//     PlcTask Inputs/GVL_iXlinker.EtherCAT_Master_EJxxxx.Beckhoff_EJ3xxx.A_0016_EJ3202_0000_0021.RTD_Inputs_Channel_2.Status/Limit_2 <-> RTD Inputs Channel 2/Status/Limit 2
//     PlcTask Inputs/GVL_iXlinker.EtherCAT_Master_EJxxxx.Beckhoff_EJ3xxx.A_0016_EJ3202_0000_0021.RTD_Inputs_Channel_1.Status/Error <-> RTD Inputs Channel 1/Status/Error
//     PlcTask Inputs/GVL_iXlinker.EtherCAT_Master_EJxxxx.Beckhoff_EJ3xxx.A_0016_EJ3202_0000_0021.RTD_Inputs_Channel_2.Status/Error <-> RTD Inputs Channel 2/Status/Error
//     PlcTask Inputs/GVL_iXlinker.EtherCAT_Master_EJxxxx.Beckhoff_EJ3xxx.A_0016_EJ3202_0000_0021.RTD_Inputs_Channel_1.Status/TxPDO_State <-> RTD Inputs Channel 1/Status/TxPDO State
//     PlcTask Inputs/GVL_iXlinker.EtherCAT_Master_EJxxxx.Beckhoff_EJ3xxx.A_0016_EJ3202_0000_0021.RTD_Inputs_Channel_2.Status/TxPDO_State <-> RTD Inputs Channel 2/Status/TxPDO State
//     PlcTask Inputs/GVL_iXlinker.EtherCAT_Master_EJxxxx.Beckhoff_EJ3xxx.A_0016_EJ3202_0000_0021.RTD_Inputs_Channel_1.Status/TxPDO_Toggle <-> RTD Inputs Channel 1/Status/TxPDO Toggle
//     PlcTask Inputs/GVL_iXlinker.EtherCAT_Master_EJxxxx.Beckhoff_EJ3xxx.A_0016_EJ3202_0000_0021.RTD_Inputs_Channel_2.Status/TxPDO_Toggle <-> RTD Inputs Channel 2/Status/TxPDO Toggle
//     PlcTask Inputs/GVL_iXlinker.EtherCAT_Master_EJxxxx.Beckhoff_EJ3xxx.A_0016_EJ3202_0000_0021.RTD_Inputs_Channel_1.Value <-> RTD Inputs Channel 1/Value
//     PlcTask Inputs/GVL_iXlinker.EtherCAT_Master_EJxxxx.Beckhoff_EJ3xxx.A_0016_EJ3202_0000_0021.RTD_Inputs_Channel_2.Value <-> RTD Inputs Channel 2/Value
//     PlcTask Inputs/GVL_iXlinker.EtherCAT_Master_EJxxxx.Beckhoff_EJ3xxx.A_0016_EJ3202_0000_0021.WcState.WcState <-> WcState/WcState
//     PlcTask Inputs/GVL_iXlinker.EtherCAT_Master_EJxxxx.Beckhoff_EJ3xxx.A_0016_EJ3202_0000_0021.WcState.InputToggle <-> WcState/InputToggle
//     PlcTask Inputs/GVL_iXlinker.EtherCAT_Master_EJxxxx.Beckhoff_EJ3xxx.A_0016_EJ3202_0000_0021.InfoData.AdsAddr <-> InfoData/AdsAddr
//     PlcTask Inputs/GVL_iXlinker.EtherCAT_Master_EJxxxx.Beckhoff_EJ3xxx.A_0016_EJ3202_0000_0021.InfoData.State <-> InfoData/State
//   PLC/PLC Instance <-> EtherCAT Master EJxxxx/Beckhoff EJ3xxx/A_0017(EJ3214-0000-0016)
//     PlcTask Inputs/GVL_iXlinker.EtherCAT_Master_EJxxxx.Beckhoff_EJ3xxx.A_0017_EJ3214_0000_0016.RTD_Inputs_Channel_1.Status/Underrange <-> RTD Inputs Channel 1/Status/Underrange
//     PlcTask Inputs/GVL_iXlinker.EtherCAT_Master_EJxxxx.Beckhoff_EJ3xxx.A_0017_EJ3214_0000_0016.RTD_Inputs_Channel_2.Status/Underrange <-> RTD Inputs Channel 2/Status/Underrange
//     PlcTask Inputs/GVL_iXlinker.EtherCAT_Master_EJxxxx.Beckhoff_EJ3xxx.A_0017_EJ3214_0000_0016.RTD_Inputs_Channel_3.Status/Underrange <-> RTD Inputs Channel 3/Status/Underrange
//     PlcTask Inputs/GVL_iXlinker.EtherCAT_Master_EJxxxx.Beckhoff_EJ3xxx.A_0017_EJ3214_0000_0016.RTD_Inputs_Channel_4.Status/Underrange <-> RTD Inputs Channel 4/Status/Underrange
//     PlcTask Inputs/GVL_iXlinker.EtherCAT_Master_EJxxxx.Beckhoff_EJ3xxx.A_0017_EJ3214_0000_0016.RTD_Inputs_Channel_1.Status/Overrange <-> RTD Inputs Channel 1/Status/Overrange
//     PlcTask Inputs/GVL_iXlinker.EtherCAT_Master_EJxxxx.Beckhoff_EJ3xxx.A_0017_EJ3214_0000_0016.RTD_Inputs_Channel_2.Status/Overrange <-> RTD Inputs Channel 2/Status/Overrange
//     PlcTask Inputs/GVL_iXlinker.EtherCAT_Master_EJxxxx.Beckhoff_EJ3xxx.A_0017_EJ3214_0000_0016.RTD_Inputs_Channel_3.Status/Overrange <-> RTD Inputs Channel 3/Status/Overrange
//     PlcTask Inputs/GVL_iXlinker.EtherCAT_Master_EJxxxx.Beckhoff_EJ3xxx.A_0017_EJ3214_0000_0016.RTD_Inputs_Channel_4.Status/Overrange <-> RTD Inputs Channel 4/Status/Overrange
//     PlcTask Inputs/GVL_iXlinker.EtherCAT_Master_EJxxxx.Beckhoff_EJ3xxx.A_0017_EJ3214_0000_0016.RTD_Inputs_Channel_1.Status/Error <-> RTD Inputs Channel 1/Status/Error
//     PlcTask Inputs/GVL_iXlinker.EtherCAT_Master_EJxxxx.Beckhoff_EJ3xxx.A_0017_EJ3214_0000_0016.RTD_Inputs_Channel_2.Status/Error <-> RTD Inputs Channel 2/Status/Error
//     PlcTask Inputs/GVL_iXlinker.EtherCAT_Master_EJxxxx.Beckhoff_EJ3xxx.A_0017_EJ3214_0000_0016.RTD_Inputs_Channel_3.Status/Error <-> RTD Inputs Channel 3/Status/Error
//     PlcTask Inputs/GVL_iXlinker.EtherCAT_Master_EJxxxx.Beckhoff_EJ3xxx.A_0017_EJ3214_0000_0016.RTD_Inputs_Channel_4.Status/Error <-> RTD Inputs Channel 4/Status/Error
//     PlcTask Inputs/GVL_iXlinker.EtherCAT_Master_EJxxxx.Beckhoff_EJ3xxx.A_0017_EJ3214_0000_0016.RTD_Inputs_Channel_1.Status/TxPDO_State <-> RTD Inputs Channel 1/Status/TxPDO State
//     PlcTask Inputs/GVL_iXlinker.EtherCAT_Master_EJxxxx.Beckhoff_EJ3xxx.A_0017_EJ3214_0000_0016.RTD_Inputs_Channel_2.Status/TxPDO_State <-> RTD Inputs Channel 2/Status/TxPDO State
//     PlcTask Inputs/GVL_iXlinker.EtherCAT_Master_EJxxxx.Beckhoff_EJ3xxx.A_0017_EJ3214_0000_0016.RTD_Inputs_Channel_3.Status/TxPDO_State <-> RTD Inputs Channel 3/Status/TxPDO State
//     PlcTask Inputs/GVL_iXlinker.EtherCAT_Master_EJxxxx.Beckhoff_EJ3xxx.A_0017_EJ3214_0000_0016.RTD_Inputs_Channel_4.Status/TxPDO_State <-> RTD Inputs Channel 4/Status/TxPDO State
//     PlcTask Inputs/GVL_iXlinker.EtherCAT_Master_EJxxxx.Beckhoff_EJ3xxx.A_0017_EJ3214_0000_0016.RTD_Inputs_Channel_1.Status/TxPDO_Toggle <-> RTD Inputs Channel 1/Status/TxPDO Toggle
//     PlcTask Inputs/GVL_iXlinker.EtherCAT_Master_EJxxxx.Beckhoff_EJ3xxx.A_0017_EJ3214_0000_0016.RTD_Inputs_Channel_2.Status/TxPDO_Toggle <-> RTD Inputs Channel 2/Status/TxPDO Toggle
//     PlcTask Inputs/GVL_iXlinker.EtherCAT_Master_EJxxxx.Beckhoff_EJ3xxx.A_0017_EJ3214_0000_0016.RTD_Inputs_Channel_3.Status/TxPDO_Toggle <-> RTD Inputs Channel 3/Status/TxPDO Toggle
//     PlcTask Inputs/GVL_iXlinker.EtherCAT_Master_EJxxxx.Beckhoff_EJ3xxx.A_0017_EJ3214_0000_0016.RTD_Inputs_Channel_4.Status/TxPDO_Toggle <-> RTD Inputs Channel 4/Status/TxPDO Toggle
//     PlcTask Inputs/GVL_iXlinker.EtherCAT_Master_EJxxxx.Beckhoff_EJ3xxx.A_0017_EJ3214_0000_0016.RTD_Inputs_Channel_1.Value <-> RTD Inputs Channel 1/Value
//     PlcTask Inputs/GVL_iXlinker.EtherCAT_Master_EJxxxx.Beckhoff_EJ3xxx.A_0017_EJ3214_0000_0016.RTD_Inputs_Channel_2.Value <-> RTD Inputs Channel 2/Value
//     PlcTask Inputs/GVL_iXlinker.EtherCAT_Master_EJxxxx.Beckhoff_EJ3xxx.A_0017_EJ3214_0000_0016.RTD_Inputs_Channel_3.Value <-> RTD Inputs Channel 3/Value
//     PlcTask Inputs/GVL_iXlinker.EtherCAT_Master_EJxxxx.Beckhoff_EJ3xxx.A_0017_EJ3214_0000_0016.RTD_Inputs_Channel_4.Value <-> RTD Inputs Channel 4/Value
//     PlcTask Inputs/GVL_iXlinker.EtherCAT_Master_EJxxxx.Beckhoff_EJ3xxx.A_0017_EJ3214_0000_0016.WcState.WcState <-> WcState/WcState
//     PlcTask Inputs/GVL_iXlinker.EtherCAT_Master_EJxxxx.Beckhoff_EJ3xxx.A_0017_EJ3214_0000_0016.WcState.InputToggle <-> WcState/InputToggle
//     PlcTask Inputs/GVL_iXlinker.EtherCAT_Master_EJxxxx.Beckhoff_EJ3xxx.A_0017_EJ3214_0000_0016.InfoData.AdsAddr <-> InfoData/AdsAddr
//     PlcTask Inputs/GVL_iXlinker.EtherCAT_Master_EJxxxx.Beckhoff_EJ3xxx.A_0017_EJ3214_0000_0016.InfoData.State <-> InfoData/State
//   PLC/PLC Instance <-> EtherCAT Master EJxxxx/Beckhoff EJ3xxx/A_0018(EJ3255-0000-0023)
//     PlcTask Inputs/GVL_iXlinker.EtherCAT_Master_EJxxxx.Beckhoff_EJ3xxx.A_0018_EJ3255_0000_0023.AI_Standard_Channel_1.Status/Underrange <-> AI Standard Channel 1/Status/Underrange
//     PlcTask Inputs/GVL_iXlinker.EtherCAT_Master_EJxxxx.Beckhoff_EJ3xxx.A_0018_EJ3255_0000_0023.AI_Standard_Channel_2.Status/Underrange <-> AI Standard Channel 2/Status/Underrange
//     PlcTask Inputs/GVL_iXlinker.EtherCAT_Master_EJxxxx.Beckhoff_EJ3xxx.A_0018_EJ3255_0000_0023.AI_Standard_Channel_3.Status/Underrange <-> AI Standard Channel 3/Status/Underrange
//     PlcTask Inputs/GVL_iXlinker.EtherCAT_Master_EJxxxx.Beckhoff_EJ3xxx.A_0018_EJ3255_0000_0023.AI_Standard_Channel_4.Status/Underrange <-> AI Standard Channel 4/Status/Underrange
//     PlcTask Inputs/GVL_iXlinker.EtherCAT_Master_EJxxxx.Beckhoff_EJ3xxx.A_0018_EJ3255_0000_0023.AI_Standard_Channel_5.Status/Underrange <-> AI Standard Channel 5/Status/Underrange
//     PlcTask Inputs/GVL_iXlinker.EtherCAT_Master_EJxxxx.Beckhoff_EJ3xxx.A_0018_EJ3255_0000_0023.AI_Standard_Channel_1.Status/Overrange <-> AI Standard Channel 1/Status/Overrange
//     PlcTask Inputs/GVL_iXlinker.EtherCAT_Master_EJxxxx.Beckhoff_EJ3xxx.A_0018_EJ3255_0000_0023.AI_Standard_Channel_2.Status/Overrange <-> AI Standard Channel 2/Status/Overrange
//     PlcTask Inputs/GVL_iXlinker.EtherCAT_Master_EJxxxx.Beckhoff_EJ3xxx.A_0018_EJ3255_0000_0023.AI_Standard_Channel_3.Status/Overrange <-> AI Standard Channel 3/Status/Overrange
//     PlcTask Inputs/GVL_iXlinker.EtherCAT_Master_EJxxxx.Beckhoff_EJ3xxx.A_0018_EJ3255_0000_0023.AI_Standard_Channel_4.Status/Overrange <-> AI Standard Channel 4/Status/Overrange
//     PlcTask Inputs/GVL_iXlinker.EtherCAT_Master_EJxxxx.Beckhoff_EJ3xxx.A_0018_EJ3255_0000_0023.AI_Standard_Channel_5.Status/Overrange <-> AI Standard Channel 5/Status/Overrange
//     PlcTask Inputs/GVL_iXlinker.EtherCAT_Master_EJxxxx.Beckhoff_EJ3xxx.A_0018_EJ3255_0000_0023.AI_Standard_Channel_1.Status/Limit_1 <-> AI Standard Channel 1/Status/Limit 1
//     PlcTask Inputs/GVL_iXlinker.EtherCAT_Master_EJxxxx.Beckhoff_EJ3xxx.A_0018_EJ3255_0000_0023.AI_Standard_Channel_1.Status/Limit_2 <-> AI Standard Channel 1/Status/Limit 2
//     PlcTask Inputs/GVL_iXlinker.EtherCAT_Master_EJxxxx.Beckhoff_EJ3xxx.A_0018_EJ3255_0000_0023.AI_Standard_Channel_2.Status/Limit_1 <-> AI Standard Channel 2/Status/Limit 1
//     PlcTask Inputs/GVL_iXlinker.EtherCAT_Master_EJxxxx.Beckhoff_EJ3xxx.A_0018_EJ3255_0000_0023.AI_Standard_Channel_2.Status/Limit_2 <-> AI Standard Channel 2/Status/Limit 2
//     PlcTask Inputs/GVL_iXlinker.EtherCAT_Master_EJxxxx.Beckhoff_EJ3xxx.A_0018_EJ3255_0000_0023.AI_Standard_Channel_3.Status/Limit_1 <-> AI Standard Channel 3/Status/Limit 1
//     PlcTask Inputs/GVL_iXlinker.EtherCAT_Master_EJxxxx.Beckhoff_EJ3xxx.A_0018_EJ3255_0000_0023.AI_Standard_Channel_3.Status/Limit_2 <-> AI Standard Channel 3/Status/Limit 2
//     PlcTask Inputs/GVL_iXlinker.EtherCAT_Master_EJxxxx.Beckhoff_EJ3xxx.A_0018_EJ3255_0000_0023.AI_Standard_Channel_4.Status/Limit_1 <-> AI Standard Channel 4/Status/Limit 1
//     PlcTask Inputs/GVL_iXlinker.EtherCAT_Master_EJxxxx.Beckhoff_EJ3xxx.A_0018_EJ3255_0000_0023.AI_Standard_Channel_4.Status/Limit_2 <-> AI Standard Channel 4/Status/Limit 2
//     PlcTask Inputs/GVL_iXlinker.EtherCAT_Master_EJxxxx.Beckhoff_EJ3xxx.A_0018_EJ3255_0000_0023.AI_Standard_Channel_5.Status/Limit_1 <-> AI Standard Channel 5/Status/Limit 1
//     PlcTask Inputs/GVL_iXlinker.EtherCAT_Master_EJxxxx.Beckhoff_EJ3xxx.A_0018_EJ3255_0000_0023.AI_Standard_Channel_5.Status/Limit_2 <-> AI Standard Channel 5/Status/Limit 2
//     PlcTask Inputs/GVL_iXlinker.EtherCAT_Master_EJxxxx.Beckhoff_EJ3xxx.A_0018_EJ3255_0000_0023.AI_Standard_Channel_1.Status/Error <-> AI Standard Channel 1/Status/Error
//     PlcTask Inputs/GVL_iXlinker.EtherCAT_Master_EJxxxx.Beckhoff_EJ3xxx.A_0018_EJ3255_0000_0023.AI_Standard_Channel_2.Status/Error <-> AI Standard Channel 2/Status/Error
//     PlcTask Inputs/GVL_iXlinker.EtherCAT_Master_EJxxxx.Beckhoff_EJ3xxx.A_0018_EJ3255_0000_0023.AI_Standard_Channel_3.Status/Error <-> AI Standard Channel 3/Status/Error
//     PlcTask Inputs/GVL_iXlinker.EtherCAT_Master_EJxxxx.Beckhoff_EJ3xxx.A_0018_EJ3255_0000_0023.AI_Standard_Channel_4.Status/Error <-> AI Standard Channel 4/Status/Error
//     PlcTask Inputs/GVL_iXlinker.EtherCAT_Master_EJxxxx.Beckhoff_EJ3xxx.A_0018_EJ3255_0000_0023.AI_Standard_Channel_5.Status/Error <-> AI Standard Channel 5/Status/Error
//     PlcTask Inputs/GVL_iXlinker.EtherCAT_Master_EJxxxx.Beckhoff_EJ3xxx.A_0018_EJ3255_0000_0023.AI_Standard_Channel_1.Status/Sync_error <-> AI Standard Channel 1/Status/Sync error
//     PlcTask Inputs/GVL_iXlinker.EtherCAT_Master_EJxxxx.Beckhoff_EJ3xxx.A_0018_EJ3255_0000_0023.AI_Standard_Channel_2.Status/Sync_error <-> AI Standard Channel 2/Status/Sync error
//     PlcTask Inputs/GVL_iXlinker.EtherCAT_Master_EJxxxx.Beckhoff_EJ3xxx.A_0018_EJ3255_0000_0023.AI_Standard_Channel_3.Status/Sync_error <-> AI Standard Channel 3/Status/Sync error
//     PlcTask Inputs/GVL_iXlinker.EtherCAT_Master_EJxxxx.Beckhoff_EJ3xxx.A_0018_EJ3255_0000_0023.AI_Standard_Channel_4.Status/Sync_error <-> AI Standard Channel 4/Status/Sync error
//     PlcTask Inputs/GVL_iXlinker.EtherCAT_Master_EJxxxx.Beckhoff_EJ3xxx.A_0018_EJ3255_0000_0023.AI_Standard_Channel_5.Status/Sync_error <-> AI Standard Channel 5/Status/Sync error
//     PlcTask Inputs/GVL_iXlinker.EtherCAT_Master_EJxxxx.Beckhoff_EJ3xxx.A_0018_EJ3255_0000_0023.AI_Standard_Channel_1.Status/TxPDO_State <-> AI Standard Channel 1/Status/TxPDO State
//     PlcTask Inputs/GVL_iXlinker.EtherCAT_Master_EJxxxx.Beckhoff_EJ3xxx.A_0018_EJ3255_0000_0023.AI_Standard_Channel_2.Status/TxPDO_State <-> AI Standard Channel 2/Status/TxPDO State
//     PlcTask Inputs/GVL_iXlinker.EtherCAT_Master_EJxxxx.Beckhoff_EJ3xxx.A_0018_EJ3255_0000_0023.AI_Standard_Channel_3.Status/TxPDO_State <-> AI Standard Channel 3/Status/TxPDO State
//     PlcTask Inputs/GVL_iXlinker.EtherCAT_Master_EJxxxx.Beckhoff_EJ3xxx.A_0018_EJ3255_0000_0023.AI_Standard_Channel_4.Status/TxPDO_State <-> AI Standard Channel 4/Status/TxPDO State
//     PlcTask Inputs/GVL_iXlinker.EtherCAT_Master_EJxxxx.Beckhoff_EJ3xxx.A_0018_EJ3255_0000_0023.AI_Standard_Channel_5.Status/TxPDO_State <-> AI Standard Channel 5/Status/TxPDO State
//     PlcTask Inputs/GVL_iXlinker.EtherCAT_Master_EJxxxx.Beckhoff_EJ3xxx.A_0018_EJ3255_0000_0023.AI_Standard_Channel_1.Status/TxPDO_Toggle <-> AI Standard Channel 1/Status/TxPDO Toggle
//     PlcTask Inputs/GVL_iXlinker.EtherCAT_Master_EJxxxx.Beckhoff_EJ3xxx.A_0018_EJ3255_0000_0023.AI_Standard_Channel_2.Status/TxPDO_Toggle <-> AI Standard Channel 2/Status/TxPDO Toggle
//     PlcTask Inputs/GVL_iXlinker.EtherCAT_Master_EJxxxx.Beckhoff_EJ3xxx.A_0018_EJ3255_0000_0023.AI_Standard_Channel_3.Status/TxPDO_Toggle <-> AI Standard Channel 3/Status/TxPDO Toggle
//     PlcTask Inputs/GVL_iXlinker.EtherCAT_Master_EJxxxx.Beckhoff_EJ3xxx.A_0018_EJ3255_0000_0023.AI_Standard_Channel_4.Status/TxPDO_Toggle <-> AI Standard Channel 4/Status/TxPDO Toggle
//     PlcTask Inputs/GVL_iXlinker.EtherCAT_Master_EJxxxx.Beckhoff_EJ3xxx.A_0018_EJ3255_0000_0023.AI_Standard_Channel_5.Status/TxPDO_Toggle <-> AI Standard Channel 5/Status/TxPDO Toggle
//     PlcTask Inputs/GVL_iXlinker.EtherCAT_Master_EJxxxx.Beckhoff_EJ3xxx.A_0018_EJ3255_0000_0023.AI_Standard_Channel_1.Value <-> AI Standard Channel 1/Value
//     PlcTask Inputs/GVL_iXlinker.EtherCAT_Master_EJxxxx.Beckhoff_EJ3xxx.A_0018_EJ3255_0000_0023.AI_Standard_Channel_2.Value <-> AI Standard Channel 2/Value
//     PlcTask Inputs/GVL_iXlinker.EtherCAT_Master_EJxxxx.Beckhoff_EJ3xxx.A_0018_EJ3255_0000_0023.AI_Standard_Channel_3.Value <-> AI Standard Channel 3/Value
//     PlcTask Inputs/GVL_iXlinker.EtherCAT_Master_EJxxxx.Beckhoff_EJ3xxx.A_0018_EJ3255_0000_0023.AI_Standard_Channel_4.Value <-> AI Standard Channel 4/Value
//     PlcTask Inputs/GVL_iXlinker.EtherCAT_Master_EJxxxx.Beckhoff_EJ3xxx.A_0018_EJ3255_0000_0023.AI_Standard_Channel_5.Value <-> AI Standard Channel 5/Value
//     PlcTask Inputs/GVL_iXlinker.EtherCAT_Master_EJxxxx.Beckhoff_EJ3xxx.A_0018_EJ3255_0000_0023.WcState.WcState <-> WcState/WcState
//     PlcTask Inputs/GVL_iXlinker.EtherCAT_Master_EJxxxx.Beckhoff_EJ3xxx.A_0018_EJ3255_0000_0023.WcState.InputToggle <-> WcState/InputToggle
//     PlcTask Inputs/GVL_iXlinker.EtherCAT_Master_EJxxxx.Beckhoff_EJ3xxx.A_0018_EJ3255_0000_0023.InfoData.AdsAddr <-> InfoData/AdsAddr
//     PlcTask Inputs/GVL_iXlinker.EtherCAT_Master_EJxxxx.Beckhoff_EJ3xxx.A_0018_EJ3255_0000_0023.InfoData.State <-> InfoData/State
//   PLC/PLC Instance <-> EtherCAT Master EJxxxx/Beckhoff EJ3xxx/A_0019(EJ3318-0000-0017)
//     PlcTask Inputs/GVL_iXlinker.EtherCAT_Master_EJxxxx.Beckhoff_EJ3xxx.A_0019_EJ3318_0000_0017.TC_Channel_1.Status/Underrange <-> TC Channel 1/Status/Underrange
//     PlcTask Inputs/GVL_iXlinker.EtherCAT_Master_EJxxxx.Beckhoff_EJ3xxx.A_0019_EJ3318_0000_0017.TC_Channel_2.Status/Underrange <-> TC Channel 2/Status/Underrange
//     PlcTask Inputs/GVL_iXlinker.EtherCAT_Master_EJxxxx.Beckhoff_EJ3xxx.A_0019_EJ3318_0000_0017.TC_Channel_3.Status/Underrange <-> TC Channel 3/Status/Underrange
//     PlcTask Inputs/GVL_iXlinker.EtherCAT_Master_EJxxxx.Beckhoff_EJ3xxx.A_0019_EJ3318_0000_0017.TC_Channel_4.Status/Underrange <-> TC Channel 4/Status/Underrange
//     PlcTask Inputs/GVL_iXlinker.EtherCAT_Master_EJxxxx.Beckhoff_EJ3xxx.A_0019_EJ3318_0000_0017.TC_Channel_5.Status/Underrange <-> TC Channel 5/Status/Underrange
//     PlcTask Inputs/GVL_iXlinker.EtherCAT_Master_EJxxxx.Beckhoff_EJ3xxx.A_0019_EJ3318_0000_0017.TC_Channel_6.Status/Underrange <-> TC Channel 6/Status/Underrange
//     PlcTask Inputs/GVL_iXlinker.EtherCAT_Master_EJxxxx.Beckhoff_EJ3xxx.A_0019_EJ3318_0000_0017.TC_Channel_7.Status/Underrange <-> TC Channel 7/Status/Underrange
//     PlcTask Inputs/GVL_iXlinker.EtherCAT_Master_EJxxxx.Beckhoff_EJ3xxx.A_0019_EJ3318_0000_0017.TC_Channel_8.Status/Underrange <-> TC Channel 8/Status/Underrange
//     PlcTask Inputs/GVL_iXlinker.EtherCAT_Master_EJxxxx.Beckhoff_EJ3xxx.A_0019_EJ3318_0000_0017.TC_Channel_1.Status/Overrange <-> TC Channel 1/Status/Overrange
//     PlcTask Inputs/GVL_iXlinker.EtherCAT_Master_EJxxxx.Beckhoff_EJ3xxx.A_0019_EJ3318_0000_0017.TC_Channel_2.Status/Overrange <-> TC Channel 2/Status/Overrange
//     PlcTask Inputs/GVL_iXlinker.EtherCAT_Master_EJxxxx.Beckhoff_EJ3xxx.A_0019_EJ3318_0000_0017.TC_Channel_3.Status/Overrange <-> TC Channel 3/Status/Overrange
//     PlcTask Inputs/GVL_iXlinker.EtherCAT_Master_EJxxxx.Beckhoff_EJ3xxx.A_0019_EJ3318_0000_0017.TC_Channel_4.Status/Overrange <-> TC Channel 4/Status/Overrange
//     PlcTask Inputs/GVL_iXlinker.EtherCAT_Master_EJxxxx.Beckhoff_EJ3xxx.A_0019_EJ3318_0000_0017.TC_Channel_5.Status/Overrange <-> TC Channel 5/Status/Overrange
//     PlcTask Inputs/GVL_iXlinker.EtherCAT_Master_EJxxxx.Beckhoff_EJ3xxx.A_0019_EJ3318_0000_0017.TC_Channel_6.Status/Overrange <-> TC Channel 6/Status/Overrange
//     PlcTask Inputs/GVL_iXlinker.EtherCAT_Master_EJxxxx.Beckhoff_EJ3xxx.A_0019_EJ3318_0000_0017.TC_Channel_7.Status/Overrange <-> TC Channel 7/Status/Overrange
//     PlcTask Inputs/GVL_iXlinker.EtherCAT_Master_EJxxxx.Beckhoff_EJ3xxx.A_0019_EJ3318_0000_0017.TC_Channel_8.Status/Overrange <-> TC Channel 8/Status/Overrange
//     PlcTask Inputs/GVL_iXlinker.EtherCAT_Master_EJxxxx.Beckhoff_EJ3xxx.A_0019_EJ3318_0000_0017.TC_Channel_1.Status/Error <-> TC Channel 1/Status/Error
//     PlcTask Inputs/GVL_iXlinker.EtherCAT_Master_EJxxxx.Beckhoff_EJ3xxx.A_0019_EJ3318_0000_0017.TC_Channel_2.Status/Error <-> TC Channel 2/Status/Error
//     PlcTask Inputs/GVL_iXlinker.EtherCAT_Master_EJxxxx.Beckhoff_EJ3xxx.A_0019_EJ3318_0000_0017.TC_Channel_3.Status/Error <-> TC Channel 3/Status/Error
//     PlcTask Inputs/GVL_iXlinker.EtherCAT_Master_EJxxxx.Beckhoff_EJ3xxx.A_0019_EJ3318_0000_0017.TC_Channel_4.Status/Error <-> TC Channel 4/Status/Error
//     PlcTask Inputs/GVL_iXlinker.EtherCAT_Master_EJxxxx.Beckhoff_EJ3xxx.A_0019_EJ3318_0000_0017.TC_Channel_5.Status/Error <-> TC Channel 5/Status/Error
//     PlcTask Inputs/GVL_iXlinker.EtherCAT_Master_EJxxxx.Beckhoff_EJ3xxx.A_0019_EJ3318_0000_0017.TC_Channel_6.Status/Error <-> TC Channel 6/Status/Error
//     PlcTask Inputs/GVL_iXlinker.EtherCAT_Master_EJxxxx.Beckhoff_EJ3xxx.A_0019_EJ3318_0000_0017.TC_Channel_7.Status/Error <-> TC Channel 7/Status/Error
//     PlcTask Inputs/GVL_iXlinker.EtherCAT_Master_EJxxxx.Beckhoff_EJ3xxx.A_0019_EJ3318_0000_0017.TC_Channel_8.Status/Error <-> TC Channel 8/Status/Error
//     PlcTask Inputs/GVL_iXlinker.EtherCAT_Master_EJxxxx.Beckhoff_EJ3xxx.A_0019_EJ3318_0000_0017.TC_Channel_1.Status/TxPDO_State <-> TC Channel 1/Status/TxPDO State
//     PlcTask Inputs/GVL_iXlinker.EtherCAT_Master_EJxxxx.Beckhoff_EJ3xxx.A_0019_EJ3318_0000_0017.TC_Channel_2.Status/TxPDO_State <-> TC Channel 2/Status/TxPDO State
//     PlcTask Inputs/GVL_iXlinker.EtherCAT_Master_EJxxxx.Beckhoff_EJ3xxx.A_0019_EJ3318_0000_0017.TC_Channel_3.Status/TxPDO_State <-> TC Channel 3/Status/TxPDO State
//     PlcTask Inputs/GVL_iXlinker.EtherCAT_Master_EJxxxx.Beckhoff_EJ3xxx.A_0019_EJ3318_0000_0017.TC_Channel_4.Status/TxPDO_State <-> TC Channel 4/Status/TxPDO State
//     PlcTask Inputs/GVL_iXlinker.EtherCAT_Master_EJxxxx.Beckhoff_EJ3xxx.A_0019_EJ3318_0000_0017.TC_Channel_5.Status/TxPDO_State <-> TC Channel 5/Status/TxPDO State
//     PlcTask Inputs/GVL_iXlinker.EtherCAT_Master_EJxxxx.Beckhoff_EJ3xxx.A_0019_EJ3318_0000_0017.TC_Channel_6.Status/TxPDO_State <-> TC Channel 6/Status/TxPDO State
//     PlcTask Inputs/GVL_iXlinker.EtherCAT_Master_EJxxxx.Beckhoff_EJ3xxx.A_0019_EJ3318_0000_0017.TC_Channel_7.Status/TxPDO_State <-> TC Channel 7/Status/TxPDO State
//     PlcTask Inputs/GVL_iXlinker.EtherCAT_Master_EJxxxx.Beckhoff_EJ3xxx.A_0019_EJ3318_0000_0017.TC_Channel_8.Status/TxPDO_State <-> TC Channel 8/Status/TxPDO State
//     PlcTask Inputs/GVL_iXlinker.EtherCAT_Master_EJxxxx.Beckhoff_EJ3xxx.A_0019_EJ3318_0000_0017.TC_Channel_1.Status/TxPDO_Toggle <-> TC Channel 1/Status/TxPDO Toggle
//     PlcTask Inputs/GVL_iXlinker.EtherCAT_Master_EJxxxx.Beckhoff_EJ3xxx.A_0019_EJ3318_0000_0017.TC_Channel_2.Status/TxPDO_Toggle <-> TC Channel 2/Status/TxPDO Toggle
//     PlcTask Inputs/GVL_iXlinker.EtherCAT_Master_EJxxxx.Beckhoff_EJ3xxx.A_0019_EJ3318_0000_0017.TC_Channel_3.Status/TxPDO_Toggle <-> TC Channel 3/Status/TxPDO Toggle
//     PlcTask Inputs/GVL_iXlinker.EtherCAT_Master_EJxxxx.Beckhoff_EJ3xxx.A_0019_EJ3318_0000_0017.TC_Channel_4.Status/TxPDO_Toggle <-> TC Channel 4/Status/TxPDO Toggle
//     PlcTask Inputs/GVL_iXlinker.EtherCAT_Master_EJxxxx.Beckhoff_EJ3xxx.A_0019_EJ3318_0000_0017.TC_Channel_5.Status/TxPDO_Toggle <-> TC Channel 5/Status/TxPDO Toggle
//     PlcTask Inputs/GVL_iXlinker.EtherCAT_Master_EJxxxx.Beckhoff_EJ3xxx.A_0019_EJ3318_0000_0017.TC_Channel_6.Status/TxPDO_Toggle <-> TC Channel 6/Status/TxPDO Toggle
//     PlcTask Inputs/GVL_iXlinker.EtherCAT_Master_EJxxxx.Beckhoff_EJ3xxx.A_0019_EJ3318_0000_0017.TC_Channel_7.Status/TxPDO_Toggle <-> TC Channel 7/Status/TxPDO Toggle
//     PlcTask Inputs/GVL_iXlinker.EtherCAT_Master_EJxxxx.Beckhoff_EJ3xxx.A_0019_EJ3318_0000_0017.TC_Channel_8.Status/TxPDO_Toggle <-> TC Channel 8/Status/TxPDO Toggle
//     PlcTask Inputs/GVL_iXlinker.EtherCAT_Master_EJxxxx.Beckhoff_EJ3xxx.A_0019_EJ3318_0000_0017.TC_Channel_1.Value <-> TC Channel 1/Value
//     PlcTask Inputs/GVL_iXlinker.EtherCAT_Master_EJxxxx.Beckhoff_EJ3xxx.A_0019_EJ3318_0000_0017.TC_Channel_2.Value <-> TC Channel 2/Value
//     PlcTask Inputs/GVL_iXlinker.EtherCAT_Master_EJxxxx.Beckhoff_EJ3xxx.A_0019_EJ3318_0000_0017.TC_Channel_3.Value <-> TC Channel 3/Value
//     PlcTask Inputs/GVL_iXlinker.EtherCAT_Master_EJxxxx.Beckhoff_EJ3xxx.A_0019_EJ3318_0000_0017.TC_Channel_4.Value <-> TC Channel 4/Value
//     PlcTask Inputs/GVL_iXlinker.EtherCAT_Master_EJxxxx.Beckhoff_EJ3xxx.A_0019_EJ3318_0000_0017.TC_Channel_5.Value <-> TC Channel 5/Value
//     PlcTask Inputs/GVL_iXlinker.EtherCAT_Master_EJxxxx.Beckhoff_EJ3xxx.A_0019_EJ3318_0000_0017.TC_Channel_6.Value <-> TC Channel 6/Value
//     PlcTask Inputs/GVL_iXlinker.EtherCAT_Master_EJxxxx.Beckhoff_EJ3xxx.A_0019_EJ3318_0000_0017.TC_Channel_7.Value <-> TC Channel 7/Value
//     PlcTask Inputs/GVL_iXlinker.EtherCAT_Master_EJxxxx.Beckhoff_EJ3xxx.A_0019_EJ3318_0000_0017.TC_Channel_8.Value <-> TC Channel 8/Value
//     PlcTask Inputs/GVL_iXlinker.EtherCAT_Master_EJxxxx.Beckhoff_EJ3xxx.A_0019_EJ3318_0000_0017.RTD_Inputs_Channel_1.Status/Underrange <-> RTD Inputs Channel 1/Status/Underrange
//     PlcTask Inputs/GVL_iXlinker.EtherCAT_Master_EJxxxx.Beckhoff_EJ3xxx.A_0019_EJ3318_0000_0017.RTD_Inputs_Channel_2.Status/Underrange <-> RTD Inputs Channel 2/Status/Underrange
//     PlcTask Inputs/GVL_iXlinker.EtherCAT_Master_EJxxxx.Beckhoff_EJ3xxx.A_0019_EJ3318_0000_0017.RTD_Inputs_Channel_1.Status/Overrange <-> RTD Inputs Channel 1/Status/Overrange
//     PlcTask Inputs/GVL_iXlinker.EtherCAT_Master_EJxxxx.Beckhoff_EJ3xxx.A_0019_EJ3318_0000_0017.RTD_Inputs_Channel_2.Status/Overrange <-> RTD Inputs Channel 2/Status/Overrange
//     PlcTask Inputs/GVL_iXlinker.EtherCAT_Master_EJxxxx.Beckhoff_EJ3xxx.A_0019_EJ3318_0000_0017.RTD_Inputs_Channel_1.Status/Error <-> RTD Inputs Channel 1/Status/Error
//     PlcTask Inputs/GVL_iXlinker.EtherCAT_Master_EJxxxx.Beckhoff_EJ3xxx.A_0019_EJ3318_0000_0017.RTD_Inputs_Channel_2.Status/Error <-> RTD Inputs Channel 2/Status/Error
//     PlcTask Inputs/GVL_iXlinker.EtherCAT_Master_EJxxxx.Beckhoff_EJ3xxx.A_0019_EJ3318_0000_0017.RTD_Inputs_Channel_1.Status/TxPDO_State <-> RTD Inputs Channel 1/Status/TxPDO State
//     PlcTask Inputs/GVL_iXlinker.EtherCAT_Master_EJxxxx.Beckhoff_EJ3xxx.A_0019_EJ3318_0000_0017.RTD_Inputs_Channel_2.Status/TxPDO_State <-> RTD Inputs Channel 2/Status/TxPDO State
//     PlcTask Inputs/GVL_iXlinker.EtherCAT_Master_EJxxxx.Beckhoff_EJ3xxx.A_0019_EJ3318_0000_0017.RTD_Inputs_Channel_1.Status/TxPDO_Toggle <-> RTD Inputs Channel 1/Status/TxPDO Toggle
//     PlcTask Inputs/GVL_iXlinker.EtherCAT_Master_EJxxxx.Beckhoff_EJ3xxx.A_0019_EJ3318_0000_0017.RTD_Inputs_Channel_2.Status/TxPDO_Toggle <-> RTD Inputs Channel 2/Status/TxPDO Toggle
//     PlcTask Inputs/GVL_iXlinker.EtherCAT_Master_EJxxxx.Beckhoff_EJ3xxx.A_0019_EJ3318_0000_0017.RTD_Inputs_Channel_1.Value <-> RTD Inputs Channel 1/Value
//     PlcTask Inputs/GVL_iXlinker.EtherCAT_Master_EJxxxx.Beckhoff_EJ3xxx.A_0019_EJ3318_0000_0017.RTD_Inputs_Channel_2.Value <-> RTD Inputs Channel 2/Value
//     PlcTask Inputs/GVL_iXlinker.EtherCAT_Master_EJxxxx.Beckhoff_EJ3xxx.A_0019_EJ3318_0000_0017.WcState.WcState <-> WcState/WcState
//     PlcTask Inputs/GVL_iXlinker.EtherCAT_Master_EJxxxx.Beckhoff_EJ3xxx.A_0019_EJ3318_0000_0017.WcState.InputToggle <-> WcState/InputToggle
//     PlcTask Inputs/GVL_iXlinker.EtherCAT_Master_EJxxxx.Beckhoff_EJ3xxx.A_0019_EJ3318_0000_0017.InfoData.AdsAddr <-> InfoData/AdsAddr
//     PlcTask Inputs/GVL_iXlinker.EtherCAT_Master_EJxxxx.Beckhoff_EJ3xxx.A_0019_EJ3318_0000_0017.InfoData.State <-> InfoData/State
//   PLC/PLC Instance <-> EtherCAT Master EJxxxx/Beckhoff EJ4xxx
//     PlcTask Inputs/GVL_iXlinker.EtherCAT_Master_EJxxxx.Beckhoff_EJ4xxx.InfoData.State <-> InfoData/State
//   PLC/PLC Instance <-> EtherCAT Master EJxxxx/Beckhoff EJ4xxx/Beckhoff EJ4xxxEK1122
//     PlcTask Inputs/GVL_iXlinker.EtherCAT_Master_EJxxxx.Beckhoff_EJ4xxx.Beckhoff_EJ4xxxEK1122.InfoData.State <-> InfoData/State
//   PLC/PLC Instance <-> EtherCAT Master EJxxxx/Beckhoff EJ4xxx/Beckhoff EJ4xxxEK1122/Beckhoff EJ4xxxsub EK1100
//     PlcTask Inputs/GVL_iXlinker.EtherCAT_Master_EJxxxx.Beckhoff_EJ4xxx.Beckhoff_EJ4xxxEK1122.Beckhoff_EJ4xxxsub_EK1100.InfoData.State <-> InfoData/State
//   PLC/PLC Instance <-> EtherCAT Master EJxxxx/Beckhoff EJ4xxx/A_0001(EJ4002-0000-0017)
//     PlcTask Outputs/GVL_iXlinker.EtherCAT_Master_EJxxxx.Beckhoff_EJ4xxx.A_0001_EJ4002_0000_0017.AO_Outputs_Channel_1.Analog_output <-> AO Outputs Channel 1/Analog output
//     PlcTask Outputs/GVL_iXlinker.EtherCAT_Master_EJxxxx.Beckhoff_EJ4xxx.A_0001_EJ4002_0000_0017.AO_Outputs_Channel_2.Analog_output <-> AO Outputs Channel 2/Analog output
//     PlcTask Inputs/GVL_iXlinker.EtherCAT_Master_EJxxxx.Beckhoff_EJ4xxx.A_0001_EJ4002_0000_0017.WcState.WcState <-> WcState/WcState
//     PlcTask Inputs/GVL_iXlinker.EtherCAT_Master_EJxxxx.Beckhoff_EJ4xxx.A_0001_EJ4002_0000_0017.InfoData.AdsAddr <-> InfoData/AdsAddr
//     PlcTask Inputs/GVL_iXlinker.EtherCAT_Master_EJxxxx.Beckhoff_EJ4xxx.A_0001_EJ4002_0000_0017.InfoData.State <-> InfoData/State
//   PLC/PLC Instance <-> EtherCAT Master EJxxxx/Beckhoff EJ4xxx/A_0002(EJ4002-0000-0018)
//     PlcTask Outputs/GVL_iXlinker.EtherCAT_Master_EJxxxx.Beckhoff_EJ4xxx.A_0002_EJ4002_0000_0018.AO_Output_Channel_1.Analog_output <-> AO Output Channel 1/Analog output
//     PlcTask Outputs/GVL_iXlinker.EtherCAT_Master_EJxxxx.Beckhoff_EJ4xxx.A_0002_EJ4002_0000_0018.AO_Output_Channel_2.Analog_output <-> AO Output Channel 2/Analog output
//     PlcTask Inputs/GVL_iXlinker.EtherCAT_Master_EJxxxx.Beckhoff_EJ4xxx.A_0002_EJ4002_0000_0018.WcState.WcState <-> WcState/WcState
//     PlcTask Inputs/GVL_iXlinker.EtherCAT_Master_EJxxxx.Beckhoff_EJ4xxx.A_0002_EJ4002_0000_0018.InfoData.AdsAddr <-> InfoData/AdsAddr
//     PlcTask Inputs/GVL_iXlinker.EtherCAT_Master_EJxxxx.Beckhoff_EJ4xxx.A_0002_EJ4002_0000_0018.InfoData.State <-> InfoData/State
//   PLC/PLC Instance <-> EtherCAT Master EJxxxx/Beckhoff EJ4xxx/A_0003(EJ4004-0000-0020)
//     PlcTask Outputs/GVL_iXlinker.EtherCAT_Master_EJxxxx.Beckhoff_EJ4xxx.A_0003_EJ4004_0000_0020.AO_Outputs_Channel_1.Analog_output <-> AO Outputs Channel 1/Analog output
//     PlcTask Outputs/GVL_iXlinker.EtherCAT_Master_EJxxxx.Beckhoff_EJ4xxx.A_0003_EJ4004_0000_0020.AO_Outputs_Channel_2.Analog_output <-> AO Outputs Channel 2/Analog output
//     PlcTask Outputs/GVL_iXlinker.EtherCAT_Master_EJxxxx.Beckhoff_EJ4xxx.A_0003_EJ4004_0000_0020.AO_Outputs_Channel_3.Analog_output <-> AO Outputs Channel 3/Analog output
//     PlcTask Outputs/GVL_iXlinker.EtherCAT_Master_EJxxxx.Beckhoff_EJ4xxx.A_0003_EJ4004_0000_0020.AO_Outputs_Channel_4.Analog_output <-> AO Outputs Channel 4/Analog output
//     PlcTask Inputs/GVL_iXlinker.EtherCAT_Master_EJxxxx.Beckhoff_EJ4xxx.A_0003_EJ4004_0000_0020.WcState.WcState <-> WcState/WcState
//     PlcTask Inputs/GVL_iXlinker.EtherCAT_Master_EJxxxx.Beckhoff_EJ4xxx.A_0003_EJ4004_0000_0020.InfoData.AdsAddr <-> InfoData/AdsAddr
//     PlcTask Inputs/GVL_iXlinker.EtherCAT_Master_EJxxxx.Beckhoff_EJ4xxx.A_0003_EJ4004_0000_0020.InfoData.State <-> InfoData/State
//   PLC/PLC Instance <-> EtherCAT Master EJxxxx/Beckhoff EJ4xxx/A_0004(EJ4008-0000-0020)
//     PlcTask Outputs/GVL_iXlinker.EtherCAT_Master_EJxxxx.Beckhoff_EJ4xxx.A_0004_EJ4008_0000_0020.AO_Outputs_Channel_1.Analog_output <-> AO Outputs Channel 1/Analog output
//     PlcTask Outputs/GVL_iXlinker.EtherCAT_Master_EJxxxx.Beckhoff_EJ4xxx.A_0004_EJ4008_0000_0020.AO_Outputs_Channel_2.Analog_output <-> AO Outputs Channel 2/Analog output
//     PlcTask Outputs/GVL_iXlinker.EtherCAT_Master_EJxxxx.Beckhoff_EJ4xxx.A_0004_EJ4008_0000_0020.AO_Outputs_Channel_3.Analog_output <-> AO Outputs Channel 3/Analog output
//     PlcTask Outputs/GVL_iXlinker.EtherCAT_Master_EJxxxx.Beckhoff_EJ4xxx.A_0004_EJ4008_0000_0020.AO_Outputs_Channel_4.Analog_output <-> AO Outputs Channel 4/Analog output
//     PlcTask Outputs/GVL_iXlinker.EtherCAT_Master_EJxxxx.Beckhoff_EJ4xxx.A_0004_EJ4008_0000_0020.AO_Outputs_Channel_5.Analog_output <-> AO Outputs Channel 5/Analog output
//     PlcTask Outputs/GVL_iXlinker.EtherCAT_Master_EJxxxx.Beckhoff_EJ4xxx.A_0004_EJ4008_0000_0020.AO_Outputs_Channel_6.Analog_output <-> AO Outputs Channel 6/Analog output
//     PlcTask Outputs/GVL_iXlinker.EtherCAT_Master_EJxxxx.Beckhoff_EJ4xxx.A_0004_EJ4008_0000_0020.AO_Outputs_Channel_7.Analog_output <-> AO Outputs Channel 7/Analog output
//     PlcTask Outputs/GVL_iXlinker.EtherCAT_Master_EJxxxx.Beckhoff_EJ4xxx.A_0004_EJ4008_0000_0020.AO_Outputs_Channel_8.Analog_output <-> AO Outputs Channel 8/Analog output
//     PlcTask Inputs/GVL_iXlinker.EtherCAT_Master_EJxxxx.Beckhoff_EJ4xxx.A_0004_EJ4008_0000_0020.WcState.WcState <-> WcState/WcState
//     PlcTask Inputs/GVL_iXlinker.EtherCAT_Master_EJxxxx.Beckhoff_EJ4xxx.A_0004_EJ4008_0000_0020.InfoData.AdsAddr <-> InfoData/AdsAddr
//     PlcTask Inputs/GVL_iXlinker.EtherCAT_Master_EJxxxx.Beckhoff_EJ4xxx.A_0004_EJ4008_0000_0020.InfoData.State <-> InfoData/State
//   PLC/PLC Instance <-> EtherCAT Master EJxxxx/Beckhoff EJ4xxx/A_0005(EJ4018-0000-0016)
//     PlcTask Outputs/GVL_iXlinker.EtherCAT_Master_EJxxxx.Beckhoff_EJ4xxx.A_0005_EJ4018_0000_0016.AO_Outputs_Channel_1.Analog_output <-> AO Outputs Channel 1/Analog output
//     PlcTask Outputs/GVL_iXlinker.EtherCAT_Master_EJxxxx.Beckhoff_EJ4xxx.A_0005_EJ4018_0000_0016.AO_Outputs_Channel_2.Analog_output <-> AO Outputs Channel 2/Analog output
//     PlcTask Outputs/GVL_iXlinker.EtherCAT_Master_EJxxxx.Beckhoff_EJ4xxx.A_0005_EJ4018_0000_0016.AO_Outputs_Channel_3.Analog_output <-> AO Outputs Channel 3/Analog output
//     PlcTask Outputs/GVL_iXlinker.EtherCAT_Master_EJxxxx.Beckhoff_EJ4xxx.A_0005_EJ4018_0000_0016.AO_Outputs_Channel_4.Analog_output <-> AO Outputs Channel 4/Analog output
//     PlcTask Outputs/GVL_iXlinker.EtherCAT_Master_EJxxxx.Beckhoff_EJ4xxx.A_0005_EJ4018_0000_0016.AO_Outputs_Channel_5.Analog_output <-> AO Outputs Channel 5/Analog output
//     PlcTask Outputs/GVL_iXlinker.EtherCAT_Master_EJxxxx.Beckhoff_EJ4xxx.A_0005_EJ4018_0000_0016.AO_Outputs_Channel_6.Analog_output <-> AO Outputs Channel 6/Analog output
//     PlcTask Outputs/GVL_iXlinker.EtherCAT_Master_EJxxxx.Beckhoff_EJ4xxx.A_0005_EJ4018_0000_0016.AO_Outputs_Channel_7.Analog_output <-> AO Outputs Channel 7/Analog output
//     PlcTask Outputs/GVL_iXlinker.EtherCAT_Master_EJxxxx.Beckhoff_EJ4xxx.A_0005_EJ4018_0000_0016.AO_Outputs_Channel_8.Analog_output <-> AO Outputs Channel 8/Analog output
//     PlcTask Inputs/GVL_iXlinker.EtherCAT_Master_EJxxxx.Beckhoff_EJ4xxx.A_0005_EJ4018_0000_0016.WcState.WcState <-> WcState/WcState
//     PlcTask Inputs/GVL_iXlinker.EtherCAT_Master_EJxxxx.Beckhoff_EJ4xxx.A_0005_EJ4018_0000_0016.InfoData.AdsAddr <-> InfoData/AdsAddr
//     PlcTask Inputs/GVL_iXlinker.EtherCAT_Master_EJxxxx.Beckhoff_EJ4xxx.A_0005_EJ4018_0000_0016.InfoData.State <-> InfoData/State
//   PLC/PLC Instance <-> EtherCAT Master EJxxxx/Beckhoff EJ4xxx/A_0006(EJ4024-0000-0020)
//     PlcTask Outputs/GVL_iXlinker.EtherCAT_Master_EJxxxx.Beckhoff_EJ4xxx.A_0006_EJ4024_0000_0020.AO_Outputs_Channel_1.Analog_output <-> AO Outputs Channel 1/Analog output
//     PlcTask Outputs/GVL_iXlinker.EtherCAT_Master_EJxxxx.Beckhoff_EJ4xxx.A_0006_EJ4024_0000_0020.AO_Outputs_Channel_2.Analog_output <-> AO Outputs Channel 2/Analog output
//     PlcTask Outputs/GVL_iXlinker.EtherCAT_Master_EJxxxx.Beckhoff_EJ4xxx.A_0006_EJ4024_0000_0020.AO_Outputs_Channel_3.Analog_output <-> AO Outputs Channel 3/Analog output
//     PlcTask Outputs/GVL_iXlinker.EtherCAT_Master_EJxxxx.Beckhoff_EJ4xxx.A_0006_EJ4024_0000_0020.AO_Outputs_Channel_4.Analog_output <-> AO Outputs Channel 4/Analog output
//     PlcTask Inputs/GVL_iXlinker.EtherCAT_Master_EJxxxx.Beckhoff_EJ4xxx.A_0006_EJ4024_0000_0020.WcState.WcState <-> WcState/WcState
//     PlcTask Inputs/GVL_iXlinker.EtherCAT_Master_EJxxxx.Beckhoff_EJ4xxx.A_0006_EJ4024_0000_0020.InfoData.AdsAddr <-> InfoData/AdsAddr
//     PlcTask Inputs/GVL_iXlinker.EtherCAT_Master_EJxxxx.Beckhoff_EJ4xxx.A_0006_EJ4024_0000_0020.InfoData.State <-> InfoData/State
//   PLC/PLC Instance <-> EtherCAT Master EJxxxx/Beckhoff EJ4xxx/A_0007(EJ4132-0000-0019)
//     PlcTask Outputs/GVL_iXlinker.EtherCAT_Master_EJxxxx.Beckhoff_EJ4xxx.A_0007_EJ4132_0000_0019.AO_Outputs_Channel_1.Analog_output <-> AO Outputs Channel 1/Analog output
//     PlcTask Outputs/GVL_iXlinker.EtherCAT_Master_EJxxxx.Beckhoff_EJ4xxx.A_0007_EJ4132_0000_0019.AO_Outputs_Channel_2.Analog_output <-> AO Outputs Channel 2/Analog output
//     PlcTask Inputs/GVL_iXlinker.EtherCAT_Master_EJxxxx.Beckhoff_EJ4xxx.A_0007_EJ4132_0000_0019.WcState.WcState <-> WcState/WcState
//     PlcTask Inputs/GVL_iXlinker.EtherCAT_Master_EJxxxx.Beckhoff_EJ4xxx.A_0007_EJ4132_0000_0019.InfoData.AdsAddr <-> InfoData/AdsAddr
//     PlcTask Inputs/GVL_iXlinker.EtherCAT_Master_EJxxxx.Beckhoff_EJ4xxx.A_0007_EJ4132_0000_0019.InfoData.State <-> InfoData/State
//   PLC/PLC Instance <-> EtherCAT Master EJxxxx/Beckhoff EJ4xxx/A_0008(EJ4134-0000-0019)
//     PlcTask Outputs/GVL_iXlinker.EtherCAT_Master_EJxxxx.Beckhoff_EJ4xxx.A_0008_EJ4134_0000_0019.AO_Output_Channel_1.Analog_output <-> AO Output Channel 1/Analog output
//     PlcTask Outputs/GVL_iXlinker.EtherCAT_Master_EJxxxx.Beckhoff_EJ4xxx.A_0008_EJ4134_0000_0019.AO_Output_Channel_2.Analog_output <-> AO Output Channel 2/Analog output
//     PlcTask Outputs/GVL_iXlinker.EtherCAT_Master_EJxxxx.Beckhoff_EJ4xxx.A_0008_EJ4134_0000_0019.AO_Output_Channel_3.Analog_output <-> AO Output Channel 3/Analog output
//     PlcTask Outputs/GVL_iXlinker.EtherCAT_Master_EJxxxx.Beckhoff_EJ4xxx.A_0008_EJ4134_0000_0019.AO_Output_Channel_4.Analog_output <-> AO Output Channel 4/Analog output
//     PlcTask Inputs/GVL_iXlinker.EtherCAT_Master_EJxxxx.Beckhoff_EJ4xxx.A_0008_EJ4134_0000_0019.WcState.WcState <-> WcState/WcState
//     PlcTask Inputs/GVL_iXlinker.EtherCAT_Master_EJxxxx.Beckhoff_EJ4xxx.A_0008_EJ4134_0000_0019.InfoData.AdsAddr <-> InfoData/AdsAddr
//     PlcTask Inputs/GVL_iXlinker.EtherCAT_Master_EJxxxx.Beckhoff_EJ4xxx.A_0008_EJ4134_0000_0019.InfoData.State <-> InfoData/State
//   PLC/PLC Instance <-> EtherCAT Master EJxxxx/Beckhoff EJ4xxx/A_0009(EJ4134-0000-0020)
//     PlcTask Outputs/GVL_iXlinker.EtherCAT_Master_EJxxxx.Beckhoff_EJ4xxx.A_0009_EJ4134_0000_0020.AO_Output_Channel_1.Analog_output <-> AO Output Channel 1/Analog output
//     PlcTask Outputs/GVL_iXlinker.EtherCAT_Master_EJxxxx.Beckhoff_EJ4xxx.A_0009_EJ4134_0000_0020.AO_Output_Channel_2.Analog_output <-> AO Output Channel 2/Analog output
//     PlcTask Outputs/GVL_iXlinker.EtherCAT_Master_EJxxxx.Beckhoff_EJ4xxx.A_0009_EJ4134_0000_0020.AO_Output_Channel_3.Analog_output <-> AO Output Channel 3/Analog output
//     PlcTask Outputs/GVL_iXlinker.EtherCAT_Master_EJxxxx.Beckhoff_EJ4xxx.A_0009_EJ4134_0000_0020.AO_Output_Channel_4.Analog_output <-> AO Output Channel 4/Analog output
//     PlcTask Inputs/GVL_iXlinker.EtherCAT_Master_EJxxxx.Beckhoff_EJ4xxx.A_0009_EJ4134_0000_0020.WcState.WcState <-> WcState/WcState
//     PlcTask Inputs/GVL_iXlinker.EtherCAT_Master_EJxxxx.Beckhoff_EJ4xxx.A_0009_EJ4134_0000_0020.InfoData.AdsAddr <-> InfoData/AdsAddr
//     PlcTask Inputs/GVL_iXlinker.EtherCAT_Master_EJxxxx.Beckhoff_EJ4xxx.A_0009_EJ4134_0000_0020.InfoData.State <-> InfoData/State
//   PLC/PLC Instance <-> EtherCAT Master EJxxxx/Beckhoff EJ5xxx
//     PlcTask Inputs/GVL_iXlinker.EtherCAT_Master_EJxxxx.Beckhoff_EJ5xxx.InfoData.State <-> InfoData/State
//   PLC/PLC Instance <-> EtherCAT Master EJxxxx/Beckhoff EJ5xxx/Beckhoff EJ5xxxEK1122
//     PlcTask Inputs/GVL_iXlinker.EtherCAT_Master_EJxxxx.Beckhoff_EJ5xxx.Beckhoff_EJ5xxxEK1122.InfoData.State <-> InfoData/State
//   PLC/PLC Instance <-> EtherCAT Master EJxxxx/Beckhoff EJ5xxx/Beckhoff EJ5xxxEK1122/Beckhoff EJ5xxxsub EK1100
//     PlcTask Inputs/GVL_iXlinker.EtherCAT_Master_EJxxxx.Beckhoff_EJ5xxx.Beckhoff_EJ5xxxEK1122.Beckhoff_EJ5xxxsub_EK1100.InfoData.State <-> InfoData/State
//   PLC/PLC Instance <-> EtherCAT Master EJxxxx/Beckhoff EJ5xxx/A_0001(EJ5002-0000-0016)
//     PlcTask Inputs/GVL_iXlinker.EtherCAT_Master_EJxxxx.Beckhoff_EJ5xxx.A_0001_EJ5002_0000_0016.SSI_Inputs_Channel_1.Status/Data_error <-> SSI Inputs Channel 1/Status/Data error
//     PlcTask Inputs/GVL_iXlinker.EtherCAT_Master_EJxxxx.Beckhoff_EJ5xxx.A_0001_EJ5002_0000_0016.SSI_Inputs_Channel_2.Status/Data_error <-> SSI Inputs Channel 2/Status/Data error
//     PlcTask Inputs/GVL_iXlinker.EtherCAT_Master_EJxxxx.Beckhoff_EJ5xxx.A_0001_EJ5002_0000_0016.SSI_Inputs_Channel_1.Status/Frame_error <-> SSI Inputs Channel 1/Status/Frame error
//     PlcTask Inputs/GVL_iXlinker.EtherCAT_Master_EJxxxx.Beckhoff_EJ5xxx.A_0001_EJ5002_0000_0016.SSI_Inputs_Channel_2.Status/Frame_error <-> SSI Inputs Channel 2/Status/Frame error
//     PlcTask Inputs/GVL_iXlinker.EtherCAT_Master_EJxxxx.Beckhoff_EJ5xxx.A_0001_EJ5002_0000_0016.SSI_Inputs_Channel_1.Status/Power_failure <-> SSI Inputs Channel 1/Status/Power failure
//     PlcTask Inputs/GVL_iXlinker.EtherCAT_Master_EJxxxx.Beckhoff_EJ5xxx.A_0001_EJ5002_0000_0016.SSI_Inputs_Channel_2.Status/Power_failure <-> SSI Inputs Channel 2/Status/Power failure
//     PlcTask Inputs/GVL_iXlinker.EtherCAT_Master_EJxxxx.Beckhoff_EJ5xxx.A_0001_EJ5002_0000_0016.SSI_Inputs_Channel_1.Status/Sync_error <-> SSI Inputs Channel 1/Status/Sync error
//     PlcTask Inputs/GVL_iXlinker.EtherCAT_Master_EJxxxx.Beckhoff_EJ5xxx.A_0001_EJ5002_0000_0016.SSI_Inputs_Channel_2.Status/Sync_error <-> SSI Inputs Channel 2/Status/Sync error
//     PlcTask Inputs/GVL_iXlinker.EtherCAT_Master_EJxxxx.Beckhoff_EJ5xxx.A_0001_EJ5002_0000_0016.SSI_Inputs_Channel_1.Status/TxPDO_State <-> SSI Inputs Channel 1/Status/TxPDO State
//     PlcTask Inputs/GVL_iXlinker.EtherCAT_Master_EJxxxx.Beckhoff_EJ5xxx.A_0001_EJ5002_0000_0016.SSI_Inputs_Channel_2.Status/TxPDO_State <-> SSI Inputs Channel 2/Status/TxPDO State
//     PlcTask Inputs/GVL_iXlinker.EtherCAT_Master_EJxxxx.Beckhoff_EJ5xxx.A_0001_EJ5002_0000_0016.SSI_Inputs_Channel_1.Status/TxPDO_Toggle <-> SSI Inputs Channel 1/Status/TxPDO Toggle
//     PlcTask Inputs/GVL_iXlinker.EtherCAT_Master_EJxxxx.Beckhoff_EJ5xxx.A_0001_EJ5002_0000_0016.SSI_Inputs_Channel_2.Status/TxPDO_Toggle <-> SSI Inputs Channel 2/Status/TxPDO Toggle
//     PlcTask Inputs/GVL_iXlinker.EtherCAT_Master_EJxxxx.Beckhoff_EJ5xxx.A_0001_EJ5002_0000_0016.SSI_Inputs_Channel_1.Counter_value <-> SSI Inputs Channel 1/Counter value
//     PlcTask Inputs/GVL_iXlinker.EtherCAT_Master_EJxxxx.Beckhoff_EJ5xxx.A_0001_EJ5002_0000_0016.SSI_Inputs_Channel_2.Counter_value <-> SSI Inputs Channel 2/Counter value
//     PlcTask Inputs/GVL_iXlinker.EtherCAT_Master_EJxxxx.Beckhoff_EJ5xxx.A_0001_EJ5002_0000_0016.WcState.WcState <-> WcState/WcState
//     PlcTask Inputs/GVL_iXlinker.EtherCAT_Master_EJxxxx.Beckhoff_EJ5xxx.A_0001_EJ5002_0000_0016.WcState.InputToggle <-> WcState/InputToggle
//     PlcTask Inputs/GVL_iXlinker.EtherCAT_Master_EJxxxx.Beckhoff_EJ5xxx.A_0001_EJ5002_0000_0016.InfoData.AdsAddr <-> InfoData/AdsAddr
//     PlcTask Inputs/GVL_iXlinker.EtherCAT_Master_EJxxxx.Beckhoff_EJ5xxx.A_0001_EJ5002_0000_0016.InfoData.State <-> InfoData/State
//   PLC/PLC Instance <-> EtherCAT Master EJxxxx/Beckhoff EJ5xxx/A_0002(EJ5002-0000-0017)
//     PlcTask Inputs/GVL_iXlinker.EtherCAT_Master_EJxxxx.Beckhoff_EJ5xxx.A_0002_EJ5002_0000_0017.SSI_Inputs_Channel_1.Status/Data_error <-> SSI Inputs Channel 1/Status/Data error
//     PlcTask Inputs/GVL_iXlinker.EtherCAT_Master_EJxxxx.Beckhoff_EJ5xxx.A_0002_EJ5002_0000_0017.SSI_Inputs_Channel_2.Status/Data_error <-> SSI Inputs Channel 2/Status/Data error
//     PlcTask Inputs/GVL_iXlinker.EtherCAT_Master_EJxxxx.Beckhoff_EJ5xxx.A_0002_EJ5002_0000_0017.SSI_Inputs_Channel_1.Status/Frame_error <-> SSI Inputs Channel 1/Status/Frame error
//     PlcTask Inputs/GVL_iXlinker.EtherCAT_Master_EJxxxx.Beckhoff_EJ5xxx.A_0002_EJ5002_0000_0017.SSI_Inputs_Channel_2.Status/Frame_error <-> SSI Inputs Channel 2/Status/Frame error
//     PlcTask Inputs/GVL_iXlinker.EtherCAT_Master_EJxxxx.Beckhoff_EJ5xxx.A_0002_EJ5002_0000_0017.SSI_Inputs_Channel_1.Status/Power_failure <-> SSI Inputs Channel 1/Status/Power failure
//     PlcTask Inputs/GVL_iXlinker.EtherCAT_Master_EJxxxx.Beckhoff_EJ5xxx.A_0002_EJ5002_0000_0017.SSI_Inputs_Channel_2.Status/Power_failure <-> SSI Inputs Channel 2/Status/Power failure
//     PlcTask Inputs/GVL_iXlinker.EtherCAT_Master_EJxxxx.Beckhoff_EJ5xxx.A_0002_EJ5002_0000_0017.SSI_Inputs_Channel_1.Status/Data_mismatch <-> SSI Inputs Channel 1/Status/Data mismatch
//     PlcTask Inputs/GVL_iXlinker.EtherCAT_Master_EJxxxx.Beckhoff_EJ5xxx.A_0002_EJ5002_0000_0017.SSI_Inputs_Channel_2.Status/Data_mismatch <-> SSI Inputs Channel 2/Status/Data mismatch
//     PlcTask Inputs/GVL_iXlinker.EtherCAT_Master_EJxxxx.Beckhoff_EJ5xxx.A_0002_EJ5002_0000_0017.SSI_Inputs_Channel_1.Status/Sync_error <-> SSI Inputs Channel 1/Status/Sync error
//     PlcTask Inputs/GVL_iXlinker.EtherCAT_Master_EJxxxx.Beckhoff_EJ5xxx.A_0002_EJ5002_0000_0017.SSI_Inputs_Channel_2.Status/Sync_error <-> SSI Inputs Channel 2/Status/Sync error
//     PlcTask Inputs/GVL_iXlinker.EtherCAT_Master_EJxxxx.Beckhoff_EJ5xxx.A_0002_EJ5002_0000_0017.SSI_Inputs_Channel_1.Status/TxPDO_State <-> SSI Inputs Channel 1/Status/TxPDO State
//     PlcTask Inputs/GVL_iXlinker.EtherCAT_Master_EJxxxx.Beckhoff_EJ5xxx.A_0002_EJ5002_0000_0017.SSI_Inputs_Channel_2.Status/TxPDO_State <-> SSI Inputs Channel 2/Status/TxPDO State
//     PlcTask Inputs/GVL_iXlinker.EtherCAT_Master_EJxxxx.Beckhoff_EJ5xxx.A_0002_EJ5002_0000_0017.SSI_Inputs_Channel_1.Status/TxPDO_Toggle <-> SSI Inputs Channel 1/Status/TxPDO Toggle
//     PlcTask Inputs/GVL_iXlinker.EtherCAT_Master_EJxxxx.Beckhoff_EJ5xxx.A_0002_EJ5002_0000_0017.SSI_Inputs_Channel_2.Status/TxPDO_Toggle <-> SSI Inputs Channel 2/Status/TxPDO Toggle
//     PlcTask Inputs/GVL_iXlinker.EtherCAT_Master_EJxxxx.Beckhoff_EJ5xxx.A_0002_EJ5002_0000_0017.SSI_Inputs_Channel_1.Counter_value <-> SSI Inputs Channel 1/Counter value
//     PlcTask Inputs/GVL_iXlinker.EtherCAT_Master_EJxxxx.Beckhoff_EJ5xxx.A_0002_EJ5002_0000_0017.SSI_Inputs_Channel_2.Counter_value <-> SSI Inputs Channel 2/Counter value
//     PlcTask Inputs/GVL_iXlinker.EtherCAT_Master_EJxxxx.Beckhoff_EJ5xxx.A_0002_EJ5002_0000_0017.WcState.WcState <-> WcState/WcState
//     PlcTask Inputs/GVL_iXlinker.EtherCAT_Master_EJxxxx.Beckhoff_EJ5xxx.A_0002_EJ5002_0000_0017.WcState.InputToggle <-> WcState/InputToggle
//     PlcTask Inputs/GVL_iXlinker.EtherCAT_Master_EJxxxx.Beckhoff_EJ5xxx.A_0002_EJ5002_0000_0017.InfoData.AdsAddr <-> InfoData/AdsAddr
//     PlcTask Inputs/GVL_iXlinker.EtherCAT_Master_EJxxxx.Beckhoff_EJ5xxx.A_0002_EJ5002_0000_0017.InfoData.State <-> InfoData/State
//   PLC/PLC Instance <-> EtherCAT Master EJxxxx/Beckhoff EJ5xxx/A_0003(EJ5101-0000-0016)
//     PlcTask Inputs/GVL_iXlinker.EtherCAT_Master_EJxxxx.Beckhoff_EJ5xxx.A_0003_EJ5101_0000_0016.ENC_Status_compact.Status/Latch_C_valid <-> ENC Status compact/Status/Latch C valid
//     PlcTask Inputs/GVL_iXlinker.EtherCAT_Master_EJxxxx.Beckhoff_EJ5xxx.A_0003_EJ5101_0000_0016.ENC_Status_compact.Status/Latch_extern_valid <-> ENC Status compact/Status/Latch extern valid
//     PlcTask Inputs/GVL_iXlinker.EtherCAT_Master_EJxxxx.Beckhoff_EJ5xxx.A_0003_EJ5101_0000_0016.ENC_Status_compact.Status/Set_counter_done <-> ENC Status compact/Status/Set counter done
//     PlcTask Inputs/GVL_iXlinker.EtherCAT_Master_EJxxxx.Beckhoff_EJ5xxx.A_0003_EJ5101_0000_0016.ENC_Status_compact.Status/Counter_underflow <-> ENC Status compact/Status/Counter underflow
//     PlcTask Inputs/GVL_iXlinker.EtherCAT_Master_EJxxxx.Beckhoff_EJ5xxx.A_0003_EJ5101_0000_0016.ENC_Status_compact.Status/Counter_overflow <-> ENC Status compact/Status/Counter overflow
//     PlcTask Inputs/GVL_iXlinker.EtherCAT_Master_EJxxxx.Beckhoff_EJ5xxx.A_0003_EJ5101_0000_0016.ENC_Status_compact.Status/Status_of_input_status <-> ENC Status compact/Status/Status of input status
//     PlcTask Inputs/GVL_iXlinker.EtherCAT_Master_EJxxxx.Beckhoff_EJ5xxx.A_0003_EJ5101_0000_0016.ENC_Status_compact.Status/Open_circuit <-> ENC Status compact/Status/Open circuit
//     PlcTask Inputs/GVL_iXlinker.EtherCAT_Master_EJxxxx.Beckhoff_EJ5xxx.A_0003_EJ5101_0000_0016.ENC_Status_compact.Status/Extrapolation_stall <-> ENC Status compact/Status/Extrapolation stall
//     PlcTask Inputs/GVL_iXlinker.EtherCAT_Master_EJxxxx.Beckhoff_EJ5xxx.A_0003_EJ5101_0000_0016.ENC_Status_compact.Status/Status_of_input_A <-> ENC Status compact/Status/Status of input A
//     PlcTask Inputs/GVL_iXlinker.EtherCAT_Master_EJxxxx.Beckhoff_EJ5xxx.A_0003_EJ5101_0000_0016.ENC_Status_compact.Status/Status_of_input_B <-> ENC Status compact/Status/Status of input B
//     PlcTask Inputs/GVL_iXlinker.EtherCAT_Master_EJxxxx.Beckhoff_EJ5xxx.A_0003_EJ5101_0000_0016.ENC_Status_compact.Status/Status_of_input_C <-> ENC Status compact/Status/Status of input C
//     PlcTask Inputs/GVL_iXlinker.EtherCAT_Master_EJxxxx.Beckhoff_EJ5xxx.A_0003_EJ5101_0000_0016.ENC_Status_compact.Status/Status_of_input_gate <-> ENC Status compact/Status/Status of input gate
//     PlcTask Inputs/GVL_iXlinker.EtherCAT_Master_EJxxxx.Beckhoff_EJ5xxx.A_0003_EJ5101_0000_0016.ENC_Status_compact.Status/Status_of_extern_latch <-> ENC Status compact/Status/Status of extern latch
//     PlcTask Inputs/GVL_iXlinker.EtherCAT_Master_EJxxxx.Beckhoff_EJ5xxx.A_0003_EJ5101_0000_0016.ENC_Status_compact.Status/Sync_error <-> ENC Status compact/Status/Sync error
//     PlcTask Inputs/GVL_iXlinker.EtherCAT_Master_EJxxxx.Beckhoff_EJ5xxx.A_0003_EJ5101_0000_0016.ENC_Status_compact.Status/TxPDO_State <-> ENC Status compact/Status/TxPDO State
//     PlcTask Inputs/GVL_iXlinker.EtherCAT_Master_EJxxxx.Beckhoff_EJ5xxx.A_0003_EJ5101_0000_0016.ENC_Status_compact.Status/TxPDO_Toggle <-> ENC Status compact/Status/TxPDO Toggle
//     PlcTask Inputs/GVL_iXlinker.EtherCAT_Master_EJxxxx.Beckhoff_EJ5xxx.A_0003_EJ5101_0000_0016.ENC_Status_compact.Counter_value <-> ENC Status compact/Counter value
//     PlcTask Inputs/GVL_iXlinker.EtherCAT_Master_EJxxxx.Beckhoff_EJ5xxx.A_0003_EJ5101_0000_0016.ENC_Status_compact.Latch_value <-> ENC Status compact/Latch value
//     PlcTask Outputs/GVL_iXlinker.EtherCAT_Master_EJxxxx.Beckhoff_EJ5xxx.A_0003_EJ5101_0000_0016.ENC_Control_compact.Control/Enable_latch_C <-> ENC Control compact/Control/Enable latch C
//     PlcTask Outputs/GVL_iXlinker.EtherCAT_Master_EJxxxx.Beckhoff_EJ5xxx.A_0003_EJ5101_0000_0016.ENC_Control_compact.Control/Enable_latch_extern_on_positive_edge <-> ENC Control compact/Control/Enable latch extern on positive edge
//     PlcTask Outputs/GVL_iXlinker.EtherCAT_Master_EJxxxx.Beckhoff_EJ5xxx.A_0003_EJ5101_0000_0016.ENC_Control_compact.Control/Set_counter <-> ENC Control compact/Control/Set counter
//     PlcTask Outputs/GVL_iXlinker.EtherCAT_Master_EJxxxx.Beckhoff_EJ5xxx.A_0003_EJ5101_0000_0016.ENC_Control_compact.Control/Enable_latch_extern_on_negative_edge <-> ENC Control compact/Control/Enable latch extern on negative edge
//     PlcTask Outputs/GVL_iXlinker.EtherCAT_Master_EJxxxx.Beckhoff_EJ5xxx.A_0003_EJ5101_0000_0016.ENC_Control_compact.Set_counter_value <-> ENC Control compact/Set counter value
//     PlcTask Inputs/GVL_iXlinker.EtherCAT_Master_EJxxxx.Beckhoff_EJ5xxx.A_0003_EJ5101_0000_0016.WcState.WcState <-> WcState/WcState
//     PlcTask Inputs/GVL_iXlinker.EtherCAT_Master_EJxxxx.Beckhoff_EJ5xxx.A_0003_EJ5101_0000_0016.WcState.InputToggle <-> WcState/InputToggle
//     PlcTask Inputs/GVL_iXlinker.EtherCAT_Master_EJxxxx.Beckhoff_EJ5xxx.A_0003_EJ5101_0000_0016.InfoData.AdsAddr <-> InfoData/AdsAddr
//     PlcTask Inputs/GVL_iXlinker.EtherCAT_Master_EJxxxx.Beckhoff_EJ5xxx.A_0003_EJ5101_0000_0016.InfoData.State <-> InfoData/State
//   PLC/PLC Instance <-> EtherCAT Master EJxxxx/Beckhoff EJ5xxx/A_0004(EJ5151-0000-0016)
//     PlcTask Inputs/GVL_iXlinker.EtherCAT_Master_EJxxxx.Beckhoff_EJ5xxx.A_0004_EJ5151_0000_0016.ENC_Inputs.Status/Latch_C_valid <-> ENC Inputs/Status/Latch C valid
//     PlcTask Inputs/GVL_iXlinker.EtherCAT_Master_EJxxxx.Beckhoff_EJ5xxx.A_0004_EJ5151_0000_0016.ENC_Inputs.Status/Latch_extern_valid <-> ENC Inputs/Status/Latch extern valid
//     PlcTask Inputs/GVL_iXlinker.EtherCAT_Master_EJxxxx.Beckhoff_EJ5xxx.A_0004_EJ5151_0000_0016.ENC_Inputs.Status/Set_counter_done <-> ENC Inputs/Status/Set counter done
//     PlcTask Inputs/GVL_iXlinker.EtherCAT_Master_EJxxxx.Beckhoff_EJ5xxx.A_0004_EJ5151_0000_0016.ENC_Inputs.Status/Extrapolation_stall <-> ENC Inputs/Status/Extrapolation stall
//     PlcTask Inputs/GVL_iXlinker.EtherCAT_Master_EJxxxx.Beckhoff_EJ5xxx.A_0004_EJ5151_0000_0016.ENC_Inputs.Status/Status_of_input_A <-> ENC Inputs/Status/Status of input A
//     PlcTask Inputs/GVL_iXlinker.EtherCAT_Master_EJxxxx.Beckhoff_EJ5xxx.A_0004_EJ5151_0000_0016.ENC_Inputs.Status/Status_of_input_B <-> ENC Inputs/Status/Status of input B
//     PlcTask Inputs/GVL_iXlinker.EtherCAT_Master_EJxxxx.Beckhoff_EJ5xxx.A_0004_EJ5151_0000_0016.ENC_Inputs.Status/Status_of_input_C <-> ENC Inputs/Status/Status of input C
//     PlcTask Inputs/GVL_iXlinker.EtherCAT_Master_EJxxxx.Beckhoff_EJ5xxx.A_0004_EJ5151_0000_0016.ENC_Inputs.Status/Status_of_extern_latch <-> ENC Inputs/Status/Status of extern latch
//     PlcTask Inputs/GVL_iXlinker.EtherCAT_Master_EJxxxx.Beckhoff_EJ5xxx.A_0004_EJ5151_0000_0016.ENC_Inputs.Status/Sync_error <-> ENC Inputs/Status/Sync error
//     PlcTask Inputs/GVL_iXlinker.EtherCAT_Master_EJxxxx.Beckhoff_EJ5xxx.A_0004_EJ5151_0000_0016.ENC_Inputs.Status/TxPDO_Toggle <-> ENC Inputs/Status/TxPDO Toggle
//     PlcTask Inputs/GVL_iXlinker.EtherCAT_Master_EJxxxx.Beckhoff_EJ5xxx.A_0004_EJ5151_0000_0016.ENC_Inputs.Counter_value <-> ENC Inputs/Counter value
//     PlcTask Inputs/GVL_iXlinker.EtherCAT_Master_EJxxxx.Beckhoff_EJ5xxx.A_0004_EJ5151_0000_0016.ENC_Inputs.Latch_value <-> ENC Inputs/Latch value
//     PlcTask Inputs/GVL_iXlinker.EtherCAT_Master_EJxxxx.Beckhoff_EJ5xxx.A_0004_EJ5151_0000_0016.ENC_Inputs_1.Period_value <-> ENC Inputs_1/Period value
//     PlcTask Outputs/GVL_iXlinker.EtherCAT_Master_EJxxxx.Beckhoff_EJ5xxx.A_0004_EJ5151_0000_0016.ENC_Outputs.Control/Enable_latch_C <-> ENC Outputs/Control/Enable latch C
//     PlcTask Outputs/GVL_iXlinker.EtherCAT_Master_EJxxxx.Beckhoff_EJ5xxx.A_0004_EJ5151_0000_0016.ENC_Outputs.Control/Enable_latch_extern_on_positive_edge <-> ENC Outputs/Control/Enable latch extern on positive edge
//     PlcTask Outputs/GVL_iXlinker.EtherCAT_Master_EJxxxx.Beckhoff_EJ5xxx.A_0004_EJ5151_0000_0016.ENC_Outputs.Control/Set_counter <-> ENC Outputs/Control/Set counter
//     PlcTask Outputs/GVL_iXlinker.EtherCAT_Master_EJxxxx.Beckhoff_EJ5xxx.A_0004_EJ5151_0000_0016.ENC_Outputs.Control/Enable_latch_extern_on_negative_edge <-> ENC Outputs/Control/Enable latch extern on negative edge
//     PlcTask Outputs/GVL_iXlinker.EtherCAT_Master_EJxxxx.Beckhoff_EJ5xxx.A_0004_EJ5151_0000_0016.ENC_Outputs.Set_counter_value <-> ENC Outputs/Set counter value
//     PlcTask Inputs/GVL_iXlinker.EtherCAT_Master_EJxxxx.Beckhoff_EJ5xxx.A_0004_EJ5151_0000_0016.WcState.WcState <-> WcState/WcState
//     PlcTask Inputs/GVL_iXlinker.EtherCAT_Master_EJxxxx.Beckhoff_EJ5xxx.A_0004_EJ5151_0000_0016.WcState.InputToggle <-> WcState/InputToggle
//     PlcTask Inputs/GVL_iXlinker.EtherCAT_Master_EJxxxx.Beckhoff_EJ5xxx.A_0004_EJ5151_0000_0016.InfoData.AdsAddr <-> InfoData/AdsAddr
//     PlcTask Inputs/GVL_iXlinker.EtherCAT_Master_EJxxxx.Beckhoff_EJ5xxx.A_0004_EJ5151_0000_0016.InfoData.State <-> InfoData/State
//   PLC/PLC Instance <-> EtherCAT Master EJxxxx/Beckhoff EJ6xxx
//     PlcTask Inputs/GVL_iXlinker.EtherCAT_Master_EJxxxx.Beckhoff_EJ6xxx.InfoData.State <-> InfoData/State
//   PLC/PLC Instance <-> EtherCAT Master EJxxxx/Beckhoff EJ6xxx/Beckhoff EJ6xxxEK1122
//     PlcTask Inputs/GVL_iXlinker.EtherCAT_Master_EJxxxx.Beckhoff_EJ6xxx.Beckhoff_EJ6xxxEK1122.InfoData.State <-> InfoData/State
//   PLC/PLC Instance <-> EtherCAT Master EJxxxx/Beckhoff EJ6xxx/Beckhoff EJ6xxxEK1122/Beckhoff EJ6xxxsub EK1100
//     PlcTask Inputs/GVL_iXlinker.EtherCAT_Master_EJxxxx.Beckhoff_EJ6xxx.Beckhoff_EJ6xxxEK1122.Beckhoff_EJ6xxxsub_EK1100.InfoData.State <-> InfoData/State
//   PLC/PLC Instance <-> EtherCAT Master EJxxxx/Beckhoff EJ6xxx/A_0001(EJ6002-0000-0016)
//     PlcTask Inputs/GVL_iXlinker.EtherCAT_Master_EJxxxx.Beckhoff_EJ6xxx.A_0001_EJ6002_0000_0016.COM_Inputs_Channel_1.Status/Transmit_accepted <-> COM Inputs Channel 1/Status/Transmit accepted
//     PlcTask Inputs/GVL_iXlinker.EtherCAT_Master_EJxxxx.Beckhoff_EJ6xxx.A_0001_EJ6002_0000_0016.COM_Inputs_Channel_2.Status/Transmit_accepted <-> COM Inputs Channel 2/Status/Transmit accepted
//     PlcTask Inputs/GVL_iXlinker.EtherCAT_Master_EJxxxx.Beckhoff_EJ6xxx.A_0001_EJ6002_0000_0016.COM_Inputs_Channel_1.Status/Receive_request <-> COM Inputs Channel 1/Status/Receive request
//     PlcTask Inputs/GVL_iXlinker.EtherCAT_Master_EJxxxx.Beckhoff_EJ6xxx.A_0001_EJ6002_0000_0016.COM_Inputs_Channel_2.Status/Receive_request <-> COM Inputs Channel 2/Status/Receive request
//     PlcTask Inputs/GVL_iXlinker.EtherCAT_Master_EJxxxx.Beckhoff_EJ6xxx.A_0001_EJ6002_0000_0016.COM_Inputs_Channel_1.Status/Init_accepted <-> COM Inputs Channel 1/Status/Init accepted
//     PlcTask Inputs/GVL_iXlinker.EtherCAT_Master_EJxxxx.Beckhoff_EJ6xxx.A_0001_EJ6002_0000_0016.COM_Inputs_Channel_2.Status/Init_accepted <-> COM Inputs Channel 2/Status/Init accepted
//     PlcTask Inputs/GVL_iXlinker.EtherCAT_Master_EJxxxx.Beckhoff_EJ6xxx.A_0001_EJ6002_0000_0016.COM_Inputs_Channel_1.Status/Buffer_full <-> COM Inputs Channel 1/Status/Buffer full
//     PlcTask Inputs/GVL_iXlinker.EtherCAT_Master_EJxxxx.Beckhoff_EJ6xxx.A_0001_EJ6002_0000_0016.COM_Inputs_Channel_2.Status/Buffer_full <-> COM Inputs Channel 2/Status/Buffer full
//     PlcTask Inputs/GVL_iXlinker.EtherCAT_Master_EJxxxx.Beckhoff_EJ6xxx.A_0001_EJ6002_0000_0016.COM_Inputs_Channel_1.Status/Parity_error <-> COM Inputs Channel 1/Status/Parity error
//     PlcTask Inputs/GVL_iXlinker.EtherCAT_Master_EJxxxx.Beckhoff_EJ6xxx.A_0001_EJ6002_0000_0016.COM_Inputs_Channel_2.Status/Parity_error <-> COM Inputs Channel 2/Status/Parity error
//     PlcTask Inputs/GVL_iXlinker.EtherCAT_Master_EJxxxx.Beckhoff_EJ6xxx.A_0001_EJ6002_0000_0016.COM_Inputs_Channel_1.Status/Framing_error <-> COM Inputs Channel 1/Status/Framing error
//     PlcTask Inputs/GVL_iXlinker.EtherCAT_Master_EJxxxx.Beckhoff_EJ6xxx.A_0001_EJ6002_0000_0016.COM_Inputs_Channel_2.Status/Framing_error <-> COM Inputs Channel 2/Status/Framing error
//     PlcTask Inputs/GVL_iXlinker.EtherCAT_Master_EJxxxx.Beckhoff_EJ6xxx.A_0001_EJ6002_0000_0016.COM_Inputs_Channel_1.Status/Overrun_error <-> COM Inputs Channel 1/Status/Overrun error
//     PlcTask Inputs/GVL_iXlinker.EtherCAT_Master_EJxxxx.Beckhoff_EJ6xxx.A_0001_EJ6002_0000_0016.COM_Inputs_Channel_2.Status/Overrun_error <-> COM Inputs Channel 2/Status/Overrun error
//     PlcTask Inputs/GVL_iXlinker.EtherCAT_Master_EJxxxx.Beckhoff_EJ6xxx.A_0001_EJ6002_0000_0016.COM_Inputs_Channel_1.Status/Input_length <-> COM Inputs Channel 1/Status/Input length
//     PlcTask Inputs/GVL_iXlinker.EtherCAT_Master_EJxxxx.Beckhoff_EJ6xxx.A_0001_EJ6002_0000_0016.COM_Inputs_Channel_2.Status/Input_length <-> COM Inputs Channel 2/Status/Input length
//     PlcTask Inputs/GVL_iXlinker.EtherCAT_Master_EJxxxx.Beckhoff_EJ6xxx.A_0001_EJ6002_0000_0016.COM_Inputs_Channel_1.Data_In[0] <-> COM Inputs Channel 1/Data In 0
//     PlcTask Inputs/GVL_iXlinker.EtherCAT_Master_EJxxxx.Beckhoff_EJ6xxx.A_0001_EJ6002_0000_0016.COM_Inputs_Channel_1.Data_In[1] <-> COM Inputs Channel 1/Data In 1
//     PlcTask Inputs/GVL_iXlinker.EtherCAT_Master_EJxxxx.Beckhoff_EJ6xxx.A_0001_EJ6002_0000_0016.COM_Inputs_Channel_1.Data_In[2] <-> COM Inputs Channel 1/Data In 2
//     PlcTask Inputs/GVL_iXlinker.EtherCAT_Master_EJxxxx.Beckhoff_EJ6xxx.A_0001_EJ6002_0000_0016.COM_Inputs_Channel_1.Data_In[3] <-> COM Inputs Channel 1/Data In 3
//     PlcTask Inputs/GVL_iXlinker.EtherCAT_Master_EJxxxx.Beckhoff_EJ6xxx.A_0001_EJ6002_0000_0016.COM_Inputs_Channel_1.Data_In[4] <-> COM Inputs Channel 1/Data In 4
//     PlcTask Inputs/GVL_iXlinker.EtherCAT_Master_EJxxxx.Beckhoff_EJ6xxx.A_0001_EJ6002_0000_0016.COM_Inputs_Channel_1.Data_In[5] <-> COM Inputs Channel 1/Data In 5
//     PlcTask Inputs/GVL_iXlinker.EtherCAT_Master_EJxxxx.Beckhoff_EJ6xxx.A_0001_EJ6002_0000_0016.COM_Inputs_Channel_1.Data_In[6] <-> COM Inputs Channel 1/Data In 6
//     PlcTask Inputs/GVL_iXlinker.EtherCAT_Master_EJxxxx.Beckhoff_EJ6xxx.A_0001_EJ6002_0000_0016.COM_Inputs_Channel_1.Data_In[7] <-> COM Inputs Channel 1/Data In 7
//     PlcTask Inputs/GVL_iXlinker.EtherCAT_Master_EJxxxx.Beckhoff_EJ6xxx.A_0001_EJ6002_0000_0016.COM_Inputs_Channel_1.Data_In[8] <-> COM Inputs Channel 1/Data In 8
//     PlcTask Inputs/GVL_iXlinker.EtherCAT_Master_EJxxxx.Beckhoff_EJ6xxx.A_0001_EJ6002_0000_0016.COM_Inputs_Channel_1.Data_In[9] <-> COM Inputs Channel 1/Data In 9
//     PlcTask Inputs/GVL_iXlinker.EtherCAT_Master_EJxxxx.Beckhoff_EJ6xxx.A_0001_EJ6002_0000_0016.COM_Inputs_Channel_1.Data_In[10] <-> COM Inputs Channel 1/Data In 10
//     PlcTask Inputs/GVL_iXlinker.EtherCAT_Master_EJxxxx.Beckhoff_EJ6xxx.A_0001_EJ6002_0000_0016.COM_Inputs_Channel_1.Data_In[11] <-> COM Inputs Channel 1/Data In 11
//     PlcTask Inputs/GVL_iXlinker.EtherCAT_Master_EJxxxx.Beckhoff_EJ6xxx.A_0001_EJ6002_0000_0016.COM_Inputs_Channel_1.Data_In[12] <-> COM Inputs Channel 1/Data In 12
//     PlcTask Inputs/GVL_iXlinker.EtherCAT_Master_EJxxxx.Beckhoff_EJ6xxx.A_0001_EJ6002_0000_0016.COM_Inputs_Channel_1.Data_In[13] <-> COM Inputs Channel 1/Data In 13
//     PlcTask Inputs/GVL_iXlinker.EtherCAT_Master_EJxxxx.Beckhoff_EJ6xxx.A_0001_EJ6002_0000_0016.COM_Inputs_Channel_1.Data_In[14] <-> COM Inputs Channel 1/Data In 14
//     PlcTask Inputs/GVL_iXlinker.EtherCAT_Master_EJxxxx.Beckhoff_EJ6xxx.A_0001_EJ6002_0000_0016.COM_Inputs_Channel_1.Data_In[15] <-> COM Inputs Channel 1/Data In 15
//     PlcTask Inputs/GVL_iXlinker.EtherCAT_Master_EJxxxx.Beckhoff_EJ6xxx.A_0001_EJ6002_0000_0016.COM_Inputs_Channel_1.Data_In[16] <-> COM Inputs Channel 1/Data In 16
//     PlcTask Inputs/GVL_iXlinker.EtherCAT_Master_EJxxxx.Beckhoff_EJ6xxx.A_0001_EJ6002_0000_0016.COM_Inputs_Channel_1.Data_In[17] <-> COM Inputs Channel 1/Data In 17
//     PlcTask Inputs/GVL_iXlinker.EtherCAT_Master_EJxxxx.Beckhoff_EJ6xxx.A_0001_EJ6002_0000_0016.COM_Inputs_Channel_1.Data_In[18] <-> COM Inputs Channel 1/Data In 18
//     PlcTask Inputs/GVL_iXlinker.EtherCAT_Master_EJxxxx.Beckhoff_EJ6xxx.A_0001_EJ6002_0000_0016.COM_Inputs_Channel_1.Data_In[19] <-> COM Inputs Channel 1/Data In 19
//     PlcTask Inputs/GVL_iXlinker.EtherCAT_Master_EJxxxx.Beckhoff_EJ6xxx.A_0001_EJ6002_0000_0016.COM_Inputs_Channel_1.Data_In[20] <-> COM Inputs Channel 1/Data In 20
//     PlcTask Inputs/GVL_iXlinker.EtherCAT_Master_EJxxxx.Beckhoff_EJ6xxx.A_0001_EJ6002_0000_0016.COM_Inputs_Channel_1.Data_In[21] <-> COM Inputs Channel 1/Data In 21
//     PlcTask Inputs/GVL_iXlinker.EtherCAT_Master_EJxxxx.Beckhoff_EJ6xxx.A_0001_EJ6002_0000_0016.COM_Inputs_Channel_2.Data_In[0] <-> COM Inputs Channel 2/Data In 0
//     PlcTask Inputs/GVL_iXlinker.EtherCAT_Master_EJxxxx.Beckhoff_EJ6xxx.A_0001_EJ6002_0000_0016.COM_Inputs_Channel_2.Data_In[1] <-> COM Inputs Channel 2/Data In 1
//     PlcTask Inputs/GVL_iXlinker.EtherCAT_Master_EJxxxx.Beckhoff_EJ6xxx.A_0001_EJ6002_0000_0016.COM_Inputs_Channel_2.Data_In[2] <-> COM Inputs Channel 2/Data In 2
//     PlcTask Inputs/GVL_iXlinker.EtherCAT_Master_EJxxxx.Beckhoff_EJ6xxx.A_0001_EJ6002_0000_0016.COM_Inputs_Channel_2.Data_In[3] <-> COM Inputs Channel 2/Data In 3
//     PlcTask Inputs/GVL_iXlinker.EtherCAT_Master_EJxxxx.Beckhoff_EJ6xxx.A_0001_EJ6002_0000_0016.COM_Inputs_Channel_2.Data_In[4] <-> COM Inputs Channel 2/Data In 4
//     PlcTask Inputs/GVL_iXlinker.EtherCAT_Master_EJxxxx.Beckhoff_EJ6xxx.A_0001_EJ6002_0000_0016.COM_Inputs_Channel_2.Data_In[5] <-> COM Inputs Channel 2/Data In 5
//     PlcTask Inputs/GVL_iXlinker.EtherCAT_Master_EJxxxx.Beckhoff_EJ6xxx.A_0001_EJ6002_0000_0016.COM_Inputs_Channel_2.Data_In[6] <-> COM Inputs Channel 2/Data In 6
//     PlcTask Inputs/GVL_iXlinker.EtherCAT_Master_EJxxxx.Beckhoff_EJ6xxx.A_0001_EJ6002_0000_0016.COM_Inputs_Channel_2.Data_In[7] <-> COM Inputs Channel 2/Data In 7
//     PlcTask Inputs/GVL_iXlinker.EtherCAT_Master_EJxxxx.Beckhoff_EJ6xxx.A_0001_EJ6002_0000_0016.COM_Inputs_Channel_2.Data_In[8] <-> COM Inputs Channel 2/Data In 8
//     PlcTask Inputs/GVL_iXlinker.EtherCAT_Master_EJxxxx.Beckhoff_EJ6xxx.A_0001_EJ6002_0000_0016.COM_Inputs_Channel_2.Data_In[9] <-> COM Inputs Channel 2/Data In 9
//     PlcTask Inputs/GVL_iXlinker.EtherCAT_Master_EJxxxx.Beckhoff_EJ6xxx.A_0001_EJ6002_0000_0016.COM_Inputs_Channel_2.Data_In[10] <-> COM Inputs Channel 2/Data In 10
//     PlcTask Inputs/GVL_iXlinker.EtherCAT_Master_EJxxxx.Beckhoff_EJ6xxx.A_0001_EJ6002_0000_0016.COM_Inputs_Channel_2.Data_In[11] <-> COM Inputs Channel 2/Data In 11
//     PlcTask Inputs/GVL_iXlinker.EtherCAT_Master_EJxxxx.Beckhoff_EJ6xxx.A_0001_EJ6002_0000_0016.COM_Inputs_Channel_2.Data_In[12] <-> COM Inputs Channel 2/Data In 12
//     PlcTask Inputs/GVL_iXlinker.EtherCAT_Master_EJxxxx.Beckhoff_EJ6xxx.A_0001_EJ6002_0000_0016.COM_Inputs_Channel_2.Data_In[13] <-> COM Inputs Channel 2/Data In 13
//     PlcTask Inputs/GVL_iXlinker.EtherCAT_Master_EJxxxx.Beckhoff_EJ6xxx.A_0001_EJ6002_0000_0016.COM_Inputs_Channel_2.Data_In[14] <-> COM Inputs Channel 2/Data In 14
//     PlcTask Inputs/GVL_iXlinker.EtherCAT_Master_EJxxxx.Beckhoff_EJ6xxx.A_0001_EJ6002_0000_0016.COM_Inputs_Channel_2.Data_In[15] <-> COM Inputs Channel 2/Data In 15
//     PlcTask Inputs/GVL_iXlinker.EtherCAT_Master_EJxxxx.Beckhoff_EJ6xxx.A_0001_EJ6002_0000_0016.COM_Inputs_Channel_2.Data_In[16] <-> COM Inputs Channel 2/Data In 16
//     PlcTask Inputs/GVL_iXlinker.EtherCAT_Master_EJxxxx.Beckhoff_EJ6xxx.A_0001_EJ6002_0000_0016.COM_Inputs_Channel_2.Data_In[17] <-> COM Inputs Channel 2/Data In 17
//     PlcTask Inputs/GVL_iXlinker.EtherCAT_Master_EJxxxx.Beckhoff_EJ6xxx.A_0001_EJ6002_0000_0016.COM_Inputs_Channel_2.Data_In[18] <-> COM Inputs Channel 2/Data In 18
//     PlcTask Inputs/GVL_iXlinker.EtherCAT_Master_EJxxxx.Beckhoff_EJ6xxx.A_0001_EJ6002_0000_0016.COM_Inputs_Channel_2.Data_In[19] <-> COM Inputs Channel 2/Data In 19
//     PlcTask Inputs/GVL_iXlinker.EtherCAT_Master_EJxxxx.Beckhoff_EJ6xxx.A_0001_EJ6002_0000_0016.COM_Inputs_Channel_2.Data_In[20] <-> COM Inputs Channel 2/Data In 20
//     PlcTask Inputs/GVL_iXlinker.EtherCAT_Master_EJxxxx.Beckhoff_EJ6xxx.A_0001_EJ6002_0000_0016.COM_Inputs_Channel_2.Data_In[21] <-> COM Inputs Channel 2/Data In 21
//     PlcTask Outputs/GVL_iXlinker.EtherCAT_Master_EJxxxx.Beckhoff_EJ6xxx.A_0001_EJ6002_0000_0016.COM_Outputs_Channel_1.Ctrl/Transmit_request <-> COM Outputs Channel 1/Ctrl/Transmit request
//     PlcTask Outputs/GVL_iXlinker.EtherCAT_Master_EJxxxx.Beckhoff_EJ6xxx.A_0001_EJ6002_0000_0016.COM_Outputs_Channel_2.Ctrl/Transmit_request <-> COM Outputs Channel 2/Ctrl/Transmit request
//     PlcTask Outputs/GVL_iXlinker.EtherCAT_Master_EJxxxx.Beckhoff_EJ6xxx.A_0001_EJ6002_0000_0016.COM_Outputs_Channel_1.Ctrl/Receive_accepted <-> COM Outputs Channel 1/Ctrl/Receive accepted
//     PlcTask Outputs/GVL_iXlinker.EtherCAT_Master_EJxxxx.Beckhoff_EJ6xxx.A_0001_EJ6002_0000_0016.COM_Outputs_Channel_2.Ctrl/Receive_accepted <-> COM Outputs Channel 2/Ctrl/Receive accepted
//     PlcTask Outputs/GVL_iXlinker.EtherCAT_Master_EJxxxx.Beckhoff_EJ6xxx.A_0001_EJ6002_0000_0016.COM_Outputs_Channel_1.Ctrl/Init_request <-> COM Outputs Channel 1/Ctrl/Init request
//     PlcTask Outputs/GVL_iXlinker.EtherCAT_Master_EJxxxx.Beckhoff_EJ6xxx.A_0001_EJ6002_0000_0016.COM_Outputs_Channel_2.Ctrl/Init_request <-> COM Outputs Channel 2/Ctrl/Init request
//     PlcTask Outputs/GVL_iXlinker.EtherCAT_Master_EJxxxx.Beckhoff_EJ6xxx.A_0001_EJ6002_0000_0016.COM_Outputs_Channel_1.Ctrl/Send_continuous <-> COM Outputs Channel 1/Ctrl/Send continuous
//     PlcTask Outputs/GVL_iXlinker.EtherCAT_Master_EJxxxx.Beckhoff_EJ6xxx.A_0001_EJ6002_0000_0016.COM_Outputs_Channel_2.Ctrl/Send_continuous <-> COM Outputs Channel 2/Ctrl/Send continuous
//     PlcTask Outputs/GVL_iXlinker.EtherCAT_Master_EJxxxx.Beckhoff_EJ6xxx.A_0001_EJ6002_0000_0016.COM_Outputs_Channel_1.Ctrl/Output_length <-> COM Outputs Channel 1/Ctrl/Output length
//     PlcTask Outputs/GVL_iXlinker.EtherCAT_Master_EJxxxx.Beckhoff_EJ6xxx.A_0001_EJ6002_0000_0016.COM_Outputs_Channel_2.Ctrl/Output_length <-> COM Outputs Channel 2/Ctrl/Output length
//     PlcTask Outputs/GVL_iXlinker.EtherCAT_Master_EJxxxx.Beckhoff_EJ6xxx.A_0001_EJ6002_0000_0016.COM_Outputs_Channel_1.Data_Out[0] <-> COM Outputs Channel 1/Data Out 0
//     PlcTask Outputs/GVL_iXlinker.EtherCAT_Master_EJxxxx.Beckhoff_EJ6xxx.A_0001_EJ6002_0000_0016.COM_Outputs_Channel_1.Data_Out[1] <-> COM Outputs Channel 1/Data Out 1
//     PlcTask Outputs/GVL_iXlinker.EtherCAT_Master_EJxxxx.Beckhoff_EJ6xxx.A_0001_EJ6002_0000_0016.COM_Outputs_Channel_1.Data_Out[2] <-> COM Outputs Channel 1/Data Out 2
//     PlcTask Outputs/GVL_iXlinker.EtherCAT_Master_EJxxxx.Beckhoff_EJ6xxx.A_0001_EJ6002_0000_0016.COM_Outputs_Channel_1.Data_Out[3] <-> COM Outputs Channel 1/Data Out 3
//     PlcTask Outputs/GVL_iXlinker.EtherCAT_Master_EJxxxx.Beckhoff_EJ6xxx.A_0001_EJ6002_0000_0016.COM_Outputs_Channel_1.Data_Out[4] <-> COM Outputs Channel 1/Data Out 4
//     PlcTask Outputs/GVL_iXlinker.EtherCAT_Master_EJxxxx.Beckhoff_EJ6xxx.A_0001_EJ6002_0000_0016.COM_Outputs_Channel_1.Data_Out[5] <-> COM Outputs Channel 1/Data Out 5
//     PlcTask Outputs/GVL_iXlinker.EtherCAT_Master_EJxxxx.Beckhoff_EJ6xxx.A_0001_EJ6002_0000_0016.COM_Outputs_Channel_1.Data_Out[6] <-> COM Outputs Channel 1/Data Out 6
//     PlcTask Outputs/GVL_iXlinker.EtherCAT_Master_EJxxxx.Beckhoff_EJ6xxx.A_0001_EJ6002_0000_0016.COM_Outputs_Channel_1.Data_Out[7] <-> COM Outputs Channel 1/Data Out 7
//     PlcTask Outputs/GVL_iXlinker.EtherCAT_Master_EJxxxx.Beckhoff_EJ6xxx.A_0001_EJ6002_0000_0016.COM_Outputs_Channel_1.Data_Out[8] <-> COM Outputs Channel 1/Data Out 8
//     PlcTask Outputs/GVL_iXlinker.EtherCAT_Master_EJxxxx.Beckhoff_EJ6xxx.A_0001_EJ6002_0000_0016.COM_Outputs_Channel_1.Data_Out[9] <-> COM Outputs Channel 1/Data Out 9
//     PlcTask Outputs/GVL_iXlinker.EtherCAT_Master_EJxxxx.Beckhoff_EJ6xxx.A_0001_EJ6002_0000_0016.COM_Outputs_Channel_1.Data_Out[10] <-> COM Outputs Channel 1/Data Out 10
//     PlcTask Outputs/GVL_iXlinker.EtherCAT_Master_EJxxxx.Beckhoff_EJ6xxx.A_0001_EJ6002_0000_0016.COM_Outputs_Channel_1.Data_Out[11] <-> COM Outputs Channel 1/Data Out 11
//     PlcTask Outputs/GVL_iXlinker.EtherCAT_Master_EJxxxx.Beckhoff_EJ6xxx.A_0001_EJ6002_0000_0016.COM_Outputs_Channel_1.Data_Out[12] <-> COM Outputs Channel 1/Data Out 12
//     PlcTask Outputs/GVL_iXlinker.EtherCAT_Master_EJxxxx.Beckhoff_EJ6xxx.A_0001_EJ6002_0000_0016.COM_Outputs_Channel_1.Data_Out[13] <-> COM Outputs Channel 1/Data Out 13
//     PlcTask Outputs/GVL_iXlinker.EtherCAT_Master_EJxxxx.Beckhoff_EJ6xxx.A_0001_EJ6002_0000_0016.COM_Outputs_Channel_1.Data_Out[14] <-> COM Outputs Channel 1/Data Out 14
//     PlcTask Outputs/GVL_iXlinker.EtherCAT_Master_EJxxxx.Beckhoff_EJ6xxx.A_0001_EJ6002_0000_0016.COM_Outputs_Channel_1.Data_Out[15] <-> COM Outputs Channel 1/Data Out 15
//     PlcTask Outputs/GVL_iXlinker.EtherCAT_Master_EJxxxx.Beckhoff_EJ6xxx.A_0001_EJ6002_0000_0016.COM_Outputs_Channel_1.Data_Out[16] <-> COM Outputs Channel 1/Data Out 16
//     PlcTask Outputs/GVL_iXlinker.EtherCAT_Master_EJxxxx.Beckhoff_EJ6xxx.A_0001_EJ6002_0000_0016.COM_Outputs_Channel_1.Data_Out[17] <-> COM Outputs Channel 1/Data Out 17
//     PlcTask Outputs/GVL_iXlinker.EtherCAT_Master_EJxxxx.Beckhoff_EJ6xxx.A_0001_EJ6002_0000_0016.COM_Outputs_Channel_1.Data_Out[18] <-> COM Outputs Channel 1/Data Out 18
//     PlcTask Outputs/GVL_iXlinker.EtherCAT_Master_EJxxxx.Beckhoff_EJ6xxx.A_0001_EJ6002_0000_0016.COM_Outputs_Channel_1.Data_Out[19] <-> COM Outputs Channel 1/Data Out 19
//     PlcTask Outputs/GVL_iXlinker.EtherCAT_Master_EJxxxx.Beckhoff_EJ6xxx.A_0001_EJ6002_0000_0016.COM_Outputs_Channel_1.Data_Out[20] <-> COM Outputs Channel 1/Data Out 20
//     PlcTask Outputs/GVL_iXlinker.EtherCAT_Master_EJxxxx.Beckhoff_EJ6xxx.A_0001_EJ6002_0000_0016.COM_Outputs_Channel_1.Data_Out[21] <-> COM Outputs Channel 1/Data Out 21
//     PlcTask Outputs/GVL_iXlinker.EtherCAT_Master_EJxxxx.Beckhoff_EJ6xxx.A_0001_EJ6002_0000_0016.COM_Outputs_Channel_2.Data_Out[0] <-> COM Outputs Channel 2/Data Out 0
//     PlcTask Outputs/GVL_iXlinker.EtherCAT_Master_EJxxxx.Beckhoff_EJ6xxx.A_0001_EJ6002_0000_0016.COM_Outputs_Channel_2.Data_Out[1] <-> COM Outputs Channel 2/Data Out 1
//     PlcTask Outputs/GVL_iXlinker.EtherCAT_Master_EJxxxx.Beckhoff_EJ6xxx.A_0001_EJ6002_0000_0016.COM_Outputs_Channel_2.Data_Out[2] <-> COM Outputs Channel 2/Data Out 2
//     PlcTask Outputs/GVL_iXlinker.EtherCAT_Master_EJxxxx.Beckhoff_EJ6xxx.A_0001_EJ6002_0000_0016.COM_Outputs_Channel_2.Data_Out[3] <-> COM Outputs Channel 2/Data Out 3
//     PlcTask Outputs/GVL_iXlinker.EtherCAT_Master_EJxxxx.Beckhoff_EJ6xxx.A_0001_EJ6002_0000_0016.COM_Outputs_Channel_2.Data_Out[4] <-> COM Outputs Channel 2/Data Out 4
//     PlcTask Outputs/GVL_iXlinker.EtherCAT_Master_EJxxxx.Beckhoff_EJ6xxx.A_0001_EJ6002_0000_0016.COM_Outputs_Channel_2.Data_Out[5] <-> COM Outputs Channel 2/Data Out 5
//     PlcTask Outputs/GVL_iXlinker.EtherCAT_Master_EJxxxx.Beckhoff_EJ6xxx.A_0001_EJ6002_0000_0016.COM_Outputs_Channel_2.Data_Out[6] <-> COM Outputs Channel 2/Data Out 6
//     PlcTask Outputs/GVL_iXlinker.EtherCAT_Master_EJxxxx.Beckhoff_EJ6xxx.A_0001_EJ6002_0000_0016.COM_Outputs_Channel_2.Data_Out[7] <-> COM Outputs Channel 2/Data Out 7
//     PlcTask Outputs/GVL_iXlinker.EtherCAT_Master_EJxxxx.Beckhoff_EJ6xxx.A_0001_EJ6002_0000_0016.COM_Outputs_Channel_2.Data_Out[8] <-> COM Outputs Channel 2/Data Out 8
//     PlcTask Outputs/GVL_iXlinker.EtherCAT_Master_EJxxxx.Beckhoff_EJ6xxx.A_0001_EJ6002_0000_0016.COM_Outputs_Channel_2.Data_Out[9] <-> COM Outputs Channel 2/Data Out 9
//     PlcTask Outputs/GVL_iXlinker.EtherCAT_Master_EJxxxx.Beckhoff_EJ6xxx.A_0001_EJ6002_0000_0016.COM_Outputs_Channel_2.Data_Out[10] <-> COM Outputs Channel 2/Data Out 10
//     PlcTask Outputs/GVL_iXlinker.EtherCAT_Master_EJxxxx.Beckhoff_EJ6xxx.A_0001_EJ6002_0000_0016.COM_Outputs_Channel_2.Data_Out[11] <-> COM Outputs Channel 2/Data Out 11
//     PlcTask Outputs/GVL_iXlinker.EtherCAT_Master_EJxxxx.Beckhoff_EJ6xxx.A_0001_EJ6002_0000_0016.COM_Outputs_Channel_2.Data_Out[12] <-> COM Outputs Channel 2/Data Out 12
//     PlcTask Outputs/GVL_iXlinker.EtherCAT_Master_EJxxxx.Beckhoff_EJ6xxx.A_0001_EJ6002_0000_0016.COM_Outputs_Channel_2.Data_Out[13] <-> COM Outputs Channel 2/Data Out 13
//     PlcTask Outputs/GVL_iXlinker.EtherCAT_Master_EJxxxx.Beckhoff_EJ6xxx.A_0001_EJ6002_0000_0016.COM_Outputs_Channel_2.Data_Out[14] <-> COM Outputs Channel 2/Data Out 14
//     PlcTask Outputs/GVL_iXlinker.EtherCAT_Master_EJxxxx.Beckhoff_EJ6xxx.A_0001_EJ6002_0000_0016.COM_Outputs_Channel_2.Data_Out[15] <-> COM Outputs Channel 2/Data Out 15
//     PlcTask Outputs/GVL_iXlinker.EtherCAT_Master_EJxxxx.Beckhoff_EJ6xxx.A_0001_EJ6002_0000_0016.COM_Outputs_Channel_2.Data_Out[16] <-> COM Outputs Channel 2/Data Out 16
//     PlcTask Outputs/GVL_iXlinker.EtherCAT_Master_EJxxxx.Beckhoff_EJ6xxx.A_0001_EJ6002_0000_0016.COM_Outputs_Channel_2.Data_Out[17] <-> COM Outputs Channel 2/Data Out 17
//     PlcTask Outputs/GVL_iXlinker.EtherCAT_Master_EJxxxx.Beckhoff_EJ6xxx.A_0001_EJ6002_0000_0016.COM_Outputs_Channel_2.Data_Out[18] <-> COM Outputs Channel 2/Data Out 18
//     PlcTask Outputs/GVL_iXlinker.EtherCAT_Master_EJxxxx.Beckhoff_EJ6xxx.A_0001_EJ6002_0000_0016.COM_Outputs_Channel_2.Data_Out[19] <-> COM Outputs Channel 2/Data Out 19
//     PlcTask Outputs/GVL_iXlinker.EtherCAT_Master_EJxxxx.Beckhoff_EJ6xxx.A_0001_EJ6002_0000_0016.COM_Outputs_Channel_2.Data_Out[20] <-> COM Outputs Channel 2/Data Out 20
//     PlcTask Outputs/GVL_iXlinker.EtherCAT_Master_EJxxxx.Beckhoff_EJ6xxx.A_0001_EJ6002_0000_0016.COM_Outputs_Channel_2.Data_Out[21] <-> COM Outputs Channel 2/Data Out 21
//     PlcTask Inputs/GVL_iXlinker.EtherCAT_Master_EJxxxx.Beckhoff_EJ6xxx.A_0001_EJ6002_0000_0016.WcState.WcState <-> WcState/WcState
//     PlcTask Inputs/GVL_iXlinker.EtherCAT_Master_EJxxxx.Beckhoff_EJ6xxx.A_0001_EJ6002_0000_0016.WcState.InputToggle <-> WcState/InputToggle
//     PlcTask Inputs/GVL_iXlinker.EtherCAT_Master_EJxxxx.Beckhoff_EJ6xxx.A_0001_EJ6002_0000_0016.InfoData.AdsAddr <-> InfoData/AdsAddr
//     PlcTask Inputs/GVL_iXlinker.EtherCAT_Master_EJxxxx.Beckhoff_EJ6xxx.A_0001_EJ6002_0000_0016.InfoData.State <-> InfoData/State
//   PLC/PLC Instance <-> EtherCAT Master EJxxxx/Beckhoff EJ6xxx/A_0002(EJ6224-0000-0016)
//     PlcTask Inputs/GVL_iXlinker.EtherCAT_Master_EJxxxx.Beckhoff_EJ6xxx.A_0002_EJ6224_0000_0016.Module_1_DeviceState_Inputs_Device.DeviceState_Inputs_Device.Device_Diag <-> Module 1 (DeviceState Inputs Device)/DeviceState Inputs Device/Device Diag
//     PlcTask Inputs/GVL_iXlinker.EtherCAT_Master_EJxxxx.Beckhoff_EJ6xxx.A_0002_EJ6224_0000_0016.Module_1_DeviceState_Inputs_Device.DeviceState_Inputs_Device.Device_State <-> Module 1 (DeviceState Inputs Device)/DeviceState Inputs Device/Device State
//     PlcTask Inputs/GVL_iXlinker.EtherCAT_Master_EJxxxx.Beckhoff_EJ6xxx.A_0002_EJ6224_0000_0016.Module_2_DeviceState_Inputs.DeviceState_Inputs.State_Ch1 <-> Module 2 (DeviceState Inputs)/DeviceState Inputs/State Ch1
//     PlcTask Inputs/GVL_iXlinker.EtherCAT_Master_EJxxxx.Beckhoff_EJ6xxx.A_0002_EJ6224_0000_0016.Module_2_DeviceState_Inputs.DeviceState_Inputs.State_Ch2 <-> Module 2 (DeviceState Inputs)/DeviceState Inputs/State Ch2
//     PlcTask Inputs/GVL_iXlinker.EtherCAT_Master_EJxxxx.Beckhoff_EJ6xxx.A_0002_EJ6224_0000_0016.Module_2_DeviceState_Inputs.DeviceState_Inputs.State_Ch3 <-> Module 2 (DeviceState Inputs)/DeviceState Inputs/State Ch3
//     PlcTask Inputs/GVL_iXlinker.EtherCAT_Master_EJxxxx.Beckhoff_EJ6xxx.A_0002_EJ6224_0000_0016.Module_2_DeviceState_Inputs.DeviceState_Inputs.State_Ch4 <-> Module 2 (DeviceState Inputs)/DeviceState Inputs/State Ch4
//     PlcTask Inputs/GVL_iXlinker.EtherCAT_Master_EJxxxx.Beckhoff_EJ6xxx.A_0002_EJ6224_0000_0016.WcState.WcState <-> WcState/WcState
//     PlcTask Inputs/GVL_iXlinker.EtherCAT_Master_EJxxxx.Beckhoff_EJ6xxx.A_0002_EJ6224_0000_0016.WcState.InputToggle <-> WcState/InputToggle
//     PlcTask Inputs/GVL_iXlinker.EtherCAT_Master_EJxxxx.Beckhoff_EJ6xxx.A_0002_EJ6224_0000_0016.InfoData.AdsAddr <-> InfoData/AdsAddr
//     PlcTask Inputs/GVL_iXlinker.EtherCAT_Master_EJxxxx.Beckhoff_EJ6xxx.A_0002_EJ6224_0000_0016.InfoData.AoeNetId <-> InfoData/AoeNetId
//     PlcTask Inputs/GVL_iXlinker.EtherCAT_Master_EJxxxx.Beckhoff_EJ6xxx.A_0002_EJ6224_0000_0016.InfoData.State <-> InfoData/State
//   PLC/PLC Instance <-> EtherCAT Master EJxxxx/Beckhoff EJ6xxx/A_0003(EJ6224-0090-0016)
//     PlcTask Inputs/GVL_iXlinker.EtherCAT_Master_EJxxxx.Beckhoff_EJ6xxx.A_0003_EJ6224_0090_0016.Module_1_DeviceState_Inputs_Device.DeviceState_Inputs_Device.Device_Diag <-> Module 1 (DeviceState Inputs Device)/DeviceState Inputs Device/Device Diag
//     PlcTask Inputs/GVL_iXlinker.EtherCAT_Master_EJxxxx.Beckhoff_EJ6xxx.A_0003_EJ6224_0090_0016.Module_1_DeviceState_Inputs_Device.DeviceState_Inputs_Device.Device_State <-> Module 1 (DeviceState Inputs Device)/DeviceState Inputs Device/Device State
//     PlcTask Inputs/GVL_iXlinker.EtherCAT_Master_EJxxxx.Beckhoff_EJ6xxx.A_0003_EJ6224_0090_0016.Module_2_DeviceState_Inputs.DeviceState_Inputs.State_Ch1 <-> Module 2 (DeviceState Inputs)/DeviceState Inputs/State Ch1
//     PlcTask Inputs/GVL_iXlinker.EtherCAT_Master_EJxxxx.Beckhoff_EJ6xxx.A_0003_EJ6224_0090_0016.Module_2_DeviceState_Inputs.DeviceState_Inputs.State_Ch2 <-> Module 2 (DeviceState Inputs)/DeviceState Inputs/State Ch2
//     PlcTask Inputs/GVL_iXlinker.EtherCAT_Master_EJxxxx.Beckhoff_EJ6xxx.A_0003_EJ6224_0090_0016.Module_2_DeviceState_Inputs.DeviceState_Inputs.State_Ch3 <-> Module 2 (DeviceState Inputs)/DeviceState Inputs/State Ch3
//     PlcTask Inputs/GVL_iXlinker.EtherCAT_Master_EJxxxx.Beckhoff_EJ6xxx.A_0003_EJ6224_0090_0016.Module_2_DeviceState_Inputs.DeviceState_Inputs.State_Ch4 <-> Module 2 (DeviceState Inputs)/DeviceState Inputs/State Ch4
//     PlcTask Inputs/GVL_iXlinker.EtherCAT_Master_EJxxxx.Beckhoff_EJ6xxx.A_0003_EJ6224_0090_0016.WcState.WcState <-> WcState/WcState
//     PlcTask Inputs/GVL_iXlinker.EtherCAT_Master_EJxxxx.Beckhoff_EJ6xxx.A_0003_EJ6224_0090_0016.WcState.InputToggle <-> WcState/InputToggle
//     PlcTask Inputs/GVL_iXlinker.EtherCAT_Master_EJxxxx.Beckhoff_EJ6xxx.A_0003_EJ6224_0090_0016.InfoData.AdsAddr <-> InfoData/AdsAddr
//     PlcTask Inputs/GVL_iXlinker.EtherCAT_Master_EJxxxx.Beckhoff_EJ6xxx.A_0003_EJ6224_0090_0016.InfoData.AoeNetId <-> InfoData/AoeNetId
//     PlcTask Inputs/GVL_iXlinker.EtherCAT_Master_EJxxxx.Beckhoff_EJ6xxx.A_0003_EJ6224_0090_0016.InfoData.State <-> InfoData/State
//   PLC/PLC Instance <-> EtherCAT Master EJxxxx/Beckhoff EJ7xxx
//     PlcTask Inputs/GVL_iXlinker.EtherCAT_Master_EJxxxx.Beckhoff_EJ7xxx.InfoData.State <-> InfoData/State
//   PLC/PLC Instance <-> EtherCAT Master EJxxxx/Beckhoff EJ7xxx/Beckhoff EJ7xxxEK1122
//     PlcTask Inputs/GVL_iXlinker.EtherCAT_Master_EJxxxx.Beckhoff_EJ7xxx.Beckhoff_EJ7xxxEK1122.InfoData.State <-> InfoData/State
//   PLC/PLC Instance <-> EtherCAT Master EJxxxx/Beckhoff EJ7xxx/Beckhoff EJ7xxxEK1122/Beckhoff EJ7xxxsub EK1100
//     PlcTask Inputs/GVL_iXlinker.EtherCAT_Master_EJxxxx.Beckhoff_EJ7xxx.Beckhoff_EJ7xxxEK1122.Beckhoff_EJ7xxxsub_EK1100.InfoData.State <-> InfoData/State
//   PLC/PLC Instance <-> EtherCAT Master EJxxxx/Beckhoff EJ7xxx/A_0001(EJ7031-0000-0026)
//     PlcTask Inputs/GVL_iXlinker.EtherCAT_Master_EJxxxx.Beckhoff_EJ7xxx.A_0001_EJ7031_0000_0026.ENC_Status_compact.Status/Latch_extern_valid <-> ENC Status compact/Status/Latch extern valid
//     PlcTask Inputs/GVL_iXlinker.EtherCAT_Master_EJxxxx.Beckhoff_EJ7xxx.A_0001_EJ7031_0000_0026.ENC_Status_compact.Status/Set_counter_done <-> ENC Status compact/Status/Set counter done
//     PlcTask Inputs/GVL_iXlinker.EtherCAT_Master_EJxxxx.Beckhoff_EJ7xxx.A_0001_EJ7031_0000_0026.ENC_Status_compact.Status/Counter_underflow <-> ENC Status compact/Status/Counter underflow
//     PlcTask Inputs/GVL_iXlinker.EtherCAT_Master_EJxxxx.Beckhoff_EJ7xxx.A_0001_EJ7031_0000_0026.ENC_Status_compact.Status/Counter_overflow <-> ENC Status compact/Status/Counter overflow
//     PlcTask Inputs/GVL_iXlinker.EtherCAT_Master_EJxxxx.Beckhoff_EJ7xxx.A_0001_EJ7031_0000_0026.ENC_Status_compact.Status/Status_of_extern_latch <-> ENC Status compact/Status/Status of extern latch
//     PlcTask Inputs/GVL_iXlinker.EtherCAT_Master_EJxxxx.Beckhoff_EJ7xxx.A_0001_EJ7031_0000_0026.ENC_Status_compact.Status/Sync_error <-> ENC Status compact/Status/Sync error
//     PlcTask Inputs/GVL_iXlinker.EtherCAT_Master_EJxxxx.Beckhoff_EJ7xxx.A_0001_EJ7031_0000_0026.ENC_Status_compact.Status/TxPDO_Toggle <-> ENC Status compact/Status/TxPDO Toggle
//     PlcTask Inputs/GVL_iXlinker.EtherCAT_Master_EJxxxx.Beckhoff_EJ7xxx.A_0001_EJ7031_0000_0026.ENC_Status_compact.Counter_value <-> ENC Status compact/Counter value
//     PlcTask Inputs/GVL_iXlinker.EtherCAT_Master_EJxxxx.Beckhoff_EJ7xxx.A_0001_EJ7031_0000_0026.ENC_Status_compact.Latch_value <-> ENC Status compact/Latch value
//     PlcTask Inputs/GVL_iXlinker.EtherCAT_Master_EJxxxx.Beckhoff_EJ7xxx.A_0001_EJ7031_0000_0026.STM_Status.Status/Ready_to_enable <-> STM Status/Status/Ready to enable
//     PlcTask Inputs/GVL_iXlinker.EtherCAT_Master_EJxxxx.Beckhoff_EJ7xxx.A_0001_EJ7031_0000_0026.STM_Status.Status/Ready <-> STM Status/Status/Ready
//     PlcTask Inputs/GVL_iXlinker.EtherCAT_Master_EJxxxx.Beckhoff_EJ7xxx.A_0001_EJ7031_0000_0026.STM_Status.Status/Warning <-> STM Status/Status/Warning
//     PlcTask Inputs/GVL_iXlinker.EtherCAT_Master_EJxxxx.Beckhoff_EJ7xxx.A_0001_EJ7031_0000_0026.STM_Status.Status/Error <-> STM Status/Status/Error
//     PlcTask Inputs/GVL_iXlinker.EtherCAT_Master_EJxxxx.Beckhoff_EJ7xxx.A_0001_EJ7031_0000_0026.STM_Status.Status/Moving_positive <-> STM Status/Status/Moving positive
//     PlcTask Inputs/GVL_iXlinker.EtherCAT_Master_EJxxxx.Beckhoff_EJ7xxx.A_0001_EJ7031_0000_0026.STM_Status.Status/Moving_negative <-> STM Status/Status/Moving negative
//     PlcTask Inputs/GVL_iXlinker.EtherCAT_Master_EJxxxx.Beckhoff_EJ7xxx.A_0001_EJ7031_0000_0026.STM_Status.Status/Torque_reduced <-> STM Status/Status/Torque reduced
//     PlcTask Inputs/GVL_iXlinker.EtherCAT_Master_EJxxxx.Beckhoff_EJ7xxx.A_0001_EJ7031_0000_0026.STM_Status.Status/Digital_input_1 <-> STM Status/Status/Digital input 1
//     PlcTask Inputs/GVL_iXlinker.EtherCAT_Master_EJxxxx.Beckhoff_EJ7xxx.A_0001_EJ7031_0000_0026.STM_Status.Status/Digital_input_2 <-> STM Status/Status/Digital input 2
//     PlcTask Inputs/GVL_iXlinker.EtherCAT_Master_EJxxxx.Beckhoff_EJ7xxx.A_0001_EJ7031_0000_0026.STM_Status.Status/Sync_error <-> STM Status/Status/Sync error
//     PlcTask Inputs/GVL_iXlinker.EtherCAT_Master_EJxxxx.Beckhoff_EJ7xxx.A_0001_EJ7031_0000_0026.STM_Status.Status/TxPDO_Toggle <-> STM Status/Status/TxPDO Toggle
//     PlcTask Outputs/GVL_iXlinker.EtherCAT_Master_EJxxxx.Beckhoff_EJ7xxx.A_0001_EJ7031_0000_0026.ENC_Control_compact.Control/Enable_latch_extern_on_positive_edge <-> ENC Control compact/Control/Enable latch extern on positive edge
//     PlcTask Outputs/GVL_iXlinker.EtherCAT_Master_EJxxxx.Beckhoff_EJ7xxx.A_0001_EJ7031_0000_0026.ENC_Control_compact.Control/Set_counter <-> ENC Control compact/Control/Set counter
//     PlcTask Outputs/GVL_iXlinker.EtherCAT_Master_EJxxxx.Beckhoff_EJ7xxx.A_0001_EJ7031_0000_0026.ENC_Control_compact.Control/Enable_latch_extern_on_negative_edge <-> ENC Control compact/Control/Enable latch extern on negative edge
//     PlcTask Outputs/GVL_iXlinker.EtherCAT_Master_EJxxxx.Beckhoff_EJ7xxx.A_0001_EJ7031_0000_0026.ENC_Control_compact.Set_counter_value <-> ENC Control compact/Set counter value
//     PlcTask Outputs/GVL_iXlinker.EtherCAT_Master_EJxxxx.Beckhoff_EJ7xxx.A_0001_EJ7031_0000_0026.STM_Control.Control/Enable <-> STM Control/Control/Enable
//     PlcTask Outputs/GVL_iXlinker.EtherCAT_Master_EJxxxx.Beckhoff_EJ7xxx.A_0001_EJ7031_0000_0026.STM_Control.Control/Reset <-> STM Control/Control/Reset
//     PlcTask Outputs/GVL_iXlinker.EtherCAT_Master_EJxxxx.Beckhoff_EJ7xxx.A_0001_EJ7031_0000_0026.STM_Control.Control/Reduce_torque <-> STM Control/Control/Reduce torque
//     PlcTask Outputs/GVL_iXlinker.EtherCAT_Master_EJxxxx.Beckhoff_EJ7xxx.A_0001_EJ7031_0000_0026.STM_Velocity.Velocity <-> STM Velocity/Velocity
//     PlcTask Inputs/GVL_iXlinker.EtherCAT_Master_EJxxxx.Beckhoff_EJ7xxx.A_0001_EJ7031_0000_0026.WcState.WcState <-> WcState/WcState
//     PlcTask Inputs/GVL_iXlinker.EtherCAT_Master_EJxxxx.Beckhoff_EJ7xxx.A_0001_EJ7031_0000_0026.WcState.InputToggle <-> WcState/InputToggle
//     PlcTask Inputs/GVL_iXlinker.EtherCAT_Master_EJxxxx.Beckhoff_EJ7xxx.A_0001_EJ7031_0000_0026.InfoData.AdsAddr <-> InfoData/AdsAddr
//     PlcTask Inputs/GVL_iXlinker.EtherCAT_Master_EJxxxx.Beckhoff_EJ7xxx.A_0001_EJ7031_0000_0026.InfoData.Chn0 <-> InfoData/Chn0
//     PlcTask Inputs/GVL_iXlinker.EtherCAT_Master_EJxxxx.Beckhoff_EJ7xxx.A_0001_EJ7031_0000_0026.InfoData.Chn1 <-> InfoData/Chn1
//     PlcTask Inputs/GVL_iXlinker.EtherCAT_Master_EJxxxx.Beckhoff_EJ7xxx.A_0001_EJ7031_0000_0026.InfoData.State <-> InfoData/State
//   PLC/PLC Instance <-> EtherCAT Master EJxxxx/Beckhoff EJ7xxx/A_0002(EJ7037-0000-0020)
//     PlcTask Inputs/GVL_iXlinker.EtherCAT_Master_EJxxxx.Beckhoff_EJ7xxx.A_0002_EJ7037_0000_0020.ENC_Status_compact.Status/Latch_C_valid <-> ENC Status compact/Status/Latch C valid
//     PlcTask Inputs/GVL_iXlinker.EtherCAT_Master_EJxxxx.Beckhoff_EJ7xxx.A_0002_EJ7037_0000_0020.ENC_Status_compact.Status/Latch_extern_valid <-> ENC Status compact/Status/Latch extern valid
//     PlcTask Inputs/GVL_iXlinker.EtherCAT_Master_EJxxxx.Beckhoff_EJ7xxx.A_0002_EJ7037_0000_0020.ENC_Status_compact.Status/Set_counter_done <-> ENC Status compact/Status/Set counter done
//     PlcTask Inputs/GVL_iXlinker.EtherCAT_Master_EJxxxx.Beckhoff_EJ7xxx.A_0002_EJ7037_0000_0020.ENC_Status_compact.Status/Counter_underflow <-> ENC Status compact/Status/Counter underflow
//     PlcTask Inputs/GVL_iXlinker.EtherCAT_Master_EJxxxx.Beckhoff_EJ7xxx.A_0002_EJ7037_0000_0020.ENC_Status_compact.Status/Counter_overflow <-> ENC Status compact/Status/Counter overflow
//     PlcTask Inputs/GVL_iXlinker.EtherCAT_Master_EJxxxx.Beckhoff_EJ7xxx.A_0002_EJ7037_0000_0020.ENC_Status_compact.Status/Extrapolation_stall <-> ENC Status compact/Status/Extrapolation stall
//     PlcTask Inputs/GVL_iXlinker.EtherCAT_Master_EJxxxx.Beckhoff_EJ7xxx.A_0002_EJ7037_0000_0020.ENC_Status_compact.Status/Status_of_input_A <-> ENC Status compact/Status/Status of input A
//     PlcTask Inputs/GVL_iXlinker.EtherCAT_Master_EJxxxx.Beckhoff_EJ7xxx.A_0002_EJ7037_0000_0020.ENC_Status_compact.Status/Status_of_input_B <-> ENC Status compact/Status/Status of input B
//     PlcTask Inputs/GVL_iXlinker.EtherCAT_Master_EJxxxx.Beckhoff_EJ7xxx.A_0002_EJ7037_0000_0020.ENC_Status_compact.Status/Status_of_input_C <-> ENC Status compact/Status/Status of input C
//     PlcTask Inputs/GVL_iXlinker.EtherCAT_Master_EJxxxx.Beckhoff_EJ7xxx.A_0002_EJ7037_0000_0020.ENC_Status_compact.Status/Status_of_extern_latch <-> ENC Status compact/Status/Status of extern latch
//     PlcTask Inputs/GVL_iXlinker.EtherCAT_Master_EJxxxx.Beckhoff_EJ7xxx.A_0002_EJ7037_0000_0020.ENC_Status_compact.Status/Sync_error <-> ENC Status compact/Status/Sync error
//     PlcTask Inputs/GVL_iXlinker.EtherCAT_Master_EJxxxx.Beckhoff_EJ7xxx.A_0002_EJ7037_0000_0020.ENC_Status_compact.Status/TxPDO_Toggle <-> ENC Status compact/Status/TxPDO Toggle
//     PlcTask Inputs/GVL_iXlinker.EtherCAT_Master_EJxxxx.Beckhoff_EJ7xxx.A_0002_EJ7037_0000_0020.ENC_Status_compact.Counter_value <-> ENC Status compact/Counter value
//     PlcTask Inputs/GVL_iXlinker.EtherCAT_Master_EJxxxx.Beckhoff_EJ7xxx.A_0002_EJ7037_0000_0020.ENC_Status_compact.Latch_value <-> ENC Status compact/Latch value
//     PlcTask Inputs/GVL_iXlinker.EtherCAT_Master_EJxxxx.Beckhoff_EJ7xxx.A_0002_EJ7037_0000_0020.STM_Status.Status/Ready_to_enable <-> STM Status/Status/Ready to enable
//     PlcTask Inputs/GVL_iXlinker.EtherCAT_Master_EJxxxx.Beckhoff_EJ7xxx.A_0002_EJ7037_0000_0020.STM_Status.Status/Ready <-> STM Status/Status/Ready
//     PlcTask Inputs/GVL_iXlinker.EtherCAT_Master_EJxxxx.Beckhoff_EJ7xxx.A_0002_EJ7037_0000_0020.STM_Status.Status/Warning <-> STM Status/Status/Warning
//     PlcTask Inputs/GVL_iXlinker.EtherCAT_Master_EJxxxx.Beckhoff_EJ7xxx.A_0002_EJ7037_0000_0020.STM_Status.Status/Error <-> STM Status/Status/Error
//     PlcTask Inputs/GVL_iXlinker.EtherCAT_Master_EJxxxx.Beckhoff_EJ7xxx.A_0002_EJ7037_0000_0020.STM_Status.Status/Moving_positive <-> STM Status/Status/Moving positive
//     PlcTask Inputs/GVL_iXlinker.EtherCAT_Master_EJxxxx.Beckhoff_EJ7xxx.A_0002_EJ7037_0000_0020.STM_Status.Status/Moving_negative <-> STM Status/Status/Moving negative
//     PlcTask Inputs/GVL_iXlinker.EtherCAT_Master_EJxxxx.Beckhoff_EJ7xxx.A_0002_EJ7037_0000_0020.STM_Status.Status/Torque_reduced <-> STM Status/Status/Torque reduced
//     PlcTask Inputs/GVL_iXlinker.EtherCAT_Master_EJxxxx.Beckhoff_EJ7xxx.A_0002_EJ7037_0000_0020.STM_Status.Status/Motor_stall <-> STM Status/Status/Motor stall
//     PlcTask Inputs/GVL_iXlinker.EtherCAT_Master_EJxxxx.Beckhoff_EJ7xxx.A_0002_EJ7037_0000_0020.STM_Status.Status/Digital_input_1 <-> STM Status/Status/Digital input 1
//     PlcTask Inputs/GVL_iXlinker.EtherCAT_Master_EJxxxx.Beckhoff_EJ7xxx.A_0002_EJ7037_0000_0020.STM_Status.Status/Digital_input_2 <-> STM Status/Status/Digital input 2
//     PlcTask Inputs/GVL_iXlinker.EtherCAT_Master_EJxxxx.Beckhoff_EJ7xxx.A_0002_EJ7037_0000_0020.STM_Status.Status/Sync_error <-> STM Status/Status/Sync error
//     PlcTask Inputs/GVL_iXlinker.EtherCAT_Master_EJxxxx.Beckhoff_EJ7xxx.A_0002_EJ7037_0000_0020.STM_Status.Status/TxPDO_Toggle <-> STM Status/Status/TxPDO Toggle
//     PlcTask Outputs/GVL_iXlinker.EtherCAT_Master_EJxxxx.Beckhoff_EJ7xxx.A_0002_EJ7037_0000_0020.ENC_Control_compact.Control/Enable_latch_C <-> ENC Control compact/Control/Enable latch C
//     PlcTask Outputs/GVL_iXlinker.EtherCAT_Master_EJxxxx.Beckhoff_EJ7xxx.A_0002_EJ7037_0000_0020.ENC_Control_compact.Control/Enable_latch_extern_on_positive_edge <-> ENC Control compact/Control/Enable latch extern on positive edge
//     PlcTask Outputs/GVL_iXlinker.EtherCAT_Master_EJxxxx.Beckhoff_EJ7xxx.A_0002_EJ7037_0000_0020.ENC_Control_compact.Control/Set_counter <-> ENC Control compact/Control/Set counter
//     PlcTask Outputs/GVL_iXlinker.EtherCAT_Master_EJxxxx.Beckhoff_EJ7xxx.A_0002_EJ7037_0000_0020.ENC_Control_compact.Control/Enable_latch_extern_on_negative_edge <-> ENC Control compact/Control/Enable latch extern on negative edge
//     PlcTask Outputs/GVL_iXlinker.EtherCAT_Master_EJxxxx.Beckhoff_EJ7xxx.A_0002_EJ7037_0000_0020.ENC_Control_compact.Set_counter_value <-> ENC Control compact/Set counter value
//     PlcTask Outputs/GVL_iXlinker.EtherCAT_Master_EJxxxx.Beckhoff_EJ7xxx.A_0002_EJ7037_0000_0020.STM_Control.Control/Enable <-> STM Control/Control/Enable
//     PlcTask Outputs/GVL_iXlinker.EtherCAT_Master_EJxxxx.Beckhoff_EJ7xxx.A_0002_EJ7037_0000_0020.STM_Control.Control/Reset <-> STM Control/Control/Reset
//     PlcTask Outputs/GVL_iXlinker.EtherCAT_Master_EJxxxx.Beckhoff_EJ7xxx.A_0002_EJ7037_0000_0020.STM_Control.Control/Reduce_torque <-> STM Control/Control/Reduce torque
//     PlcTask Outputs/GVL_iXlinker.EtherCAT_Master_EJxxxx.Beckhoff_EJ7xxx.A_0002_EJ7037_0000_0020.STM_Control.Control/Digital_output_1 <-> STM Control/Control/Digital output 1
//     PlcTask Outputs/GVL_iXlinker.EtherCAT_Master_EJxxxx.Beckhoff_EJ7xxx.A_0002_EJ7037_0000_0020.STM_Velocity.Velocity <-> STM Velocity/Velocity
//     PlcTask Inputs/GVL_iXlinker.EtherCAT_Master_EJxxxx.Beckhoff_EJ7xxx.A_0002_EJ7037_0000_0020.WcState.WcState <-> WcState/WcState
//     PlcTask Inputs/GVL_iXlinker.EtherCAT_Master_EJxxxx.Beckhoff_EJ7xxx.A_0002_EJ7037_0000_0020.WcState.InputToggle <-> WcState/InputToggle
//     PlcTask Inputs/GVL_iXlinker.EtherCAT_Master_EJxxxx.Beckhoff_EJ7xxx.A_0002_EJ7037_0000_0020.InfoData.AdsAddr <-> InfoData/AdsAddr
//     PlcTask Inputs/GVL_iXlinker.EtherCAT_Master_EJxxxx.Beckhoff_EJ7xxx.A_0002_EJ7037_0000_0020.InfoData.Chn0 <-> InfoData/Chn0
//     PlcTask Inputs/GVL_iXlinker.EtherCAT_Master_EJxxxx.Beckhoff_EJ7xxx.A_0002_EJ7037_0000_0020.InfoData.Chn1 <-> InfoData/Chn1
//     PlcTask Inputs/GVL_iXlinker.EtherCAT_Master_EJxxxx.Beckhoff_EJ7xxx.A_0002_EJ7037_0000_0020.InfoData.State <-> InfoData/State
//   PLC/PLC Instance <-> EtherCAT Master EJxxxx/Beckhoff EJ7xxx/A_0003(EJ7041-0052-0016)
//     PlcTask Inputs/GVL_iXlinker.EtherCAT_Master_EJxxxx.Beckhoff_EJ7xxx.A_0003_EJ7041_0052_0016.ENC_Status_compact.Status/Latch_extern_valid <-> ENC Status compact/Status/Latch extern valid
//     PlcTask Inputs/GVL_iXlinker.EtherCAT_Master_EJxxxx.Beckhoff_EJ7xxx.A_0003_EJ7041_0052_0016.ENC_Status_compact.Status/Set_counter_done <-> ENC Status compact/Status/Set counter done
//     PlcTask Inputs/GVL_iXlinker.EtherCAT_Master_EJxxxx.Beckhoff_EJ7xxx.A_0003_EJ7041_0052_0016.ENC_Status_compact.Status/Counter_underflow <-> ENC Status compact/Status/Counter underflow
//     PlcTask Inputs/GVL_iXlinker.EtherCAT_Master_EJxxxx.Beckhoff_EJ7xxx.A_0003_EJ7041_0052_0016.ENC_Status_compact.Status/Counter_overflow <-> ENC Status compact/Status/Counter overflow
//     PlcTask Inputs/GVL_iXlinker.EtherCAT_Master_EJxxxx.Beckhoff_EJ7xxx.A_0003_EJ7041_0052_0016.ENC_Status_compact.Status/Status_of_extern_latch <-> ENC Status compact/Status/Status of extern latch
//     PlcTask Inputs/GVL_iXlinker.EtherCAT_Master_EJxxxx.Beckhoff_EJ7xxx.A_0003_EJ7041_0052_0016.ENC_Status_compact.Status/Sync_error <-> ENC Status compact/Status/Sync error
//     PlcTask Inputs/GVL_iXlinker.EtherCAT_Master_EJxxxx.Beckhoff_EJ7xxx.A_0003_EJ7041_0052_0016.ENC_Status_compact.Status/TxPDO_Toggle <-> ENC Status compact/Status/TxPDO Toggle
//     PlcTask Inputs/GVL_iXlinker.EtherCAT_Master_EJxxxx.Beckhoff_EJ7xxx.A_0003_EJ7041_0052_0016.ENC_Status_compact.Counter_value <-> ENC Status compact/Counter value
//     PlcTask Inputs/GVL_iXlinker.EtherCAT_Master_EJxxxx.Beckhoff_EJ7xxx.A_0003_EJ7041_0052_0016.ENC_Status_compact.Latch_value <-> ENC Status compact/Latch value
//     PlcTask Inputs/GVL_iXlinker.EtherCAT_Master_EJxxxx.Beckhoff_EJ7xxx.A_0003_EJ7041_0052_0016.STM_Status.Status/Ready_to_enable <-> STM Status/Status/Ready to enable
//     PlcTask Inputs/GVL_iXlinker.EtherCAT_Master_EJxxxx.Beckhoff_EJ7xxx.A_0003_EJ7041_0052_0016.STM_Status.Status/Ready <-> STM Status/Status/Ready
//     PlcTask Inputs/GVL_iXlinker.EtherCAT_Master_EJxxxx.Beckhoff_EJ7xxx.A_0003_EJ7041_0052_0016.STM_Status.Status/Warning <-> STM Status/Status/Warning
//     PlcTask Inputs/GVL_iXlinker.EtherCAT_Master_EJxxxx.Beckhoff_EJ7xxx.A_0003_EJ7041_0052_0016.STM_Status.Status/Error <-> STM Status/Status/Error
//     PlcTask Inputs/GVL_iXlinker.EtherCAT_Master_EJxxxx.Beckhoff_EJ7xxx.A_0003_EJ7041_0052_0016.STM_Status.Status/Moving_positive <-> STM Status/Status/Moving positive
//     PlcTask Inputs/GVL_iXlinker.EtherCAT_Master_EJxxxx.Beckhoff_EJ7xxx.A_0003_EJ7041_0052_0016.STM_Status.Status/Moving_negative <-> STM Status/Status/Moving negative
//     PlcTask Inputs/GVL_iXlinker.EtherCAT_Master_EJxxxx.Beckhoff_EJ7xxx.A_0003_EJ7041_0052_0016.STM_Status.Status/Torque_reduced <-> STM Status/Status/Torque reduced
//     PlcTask Inputs/GVL_iXlinker.EtherCAT_Master_EJxxxx.Beckhoff_EJ7xxx.A_0003_EJ7041_0052_0016.STM_Status.Status/Digital_input_1 <-> STM Status/Status/Digital input 1
//     PlcTask Inputs/GVL_iXlinker.EtherCAT_Master_EJxxxx.Beckhoff_EJ7xxx.A_0003_EJ7041_0052_0016.STM_Status.Status/Digital_input_2 <-> STM Status/Status/Digital input 2
//     PlcTask Inputs/GVL_iXlinker.EtherCAT_Master_EJxxxx.Beckhoff_EJ7xxx.A_0003_EJ7041_0052_0016.STM_Status.Status/Sync_error <-> STM Status/Status/Sync error
//     PlcTask Inputs/GVL_iXlinker.EtherCAT_Master_EJxxxx.Beckhoff_EJ7xxx.A_0003_EJ7041_0052_0016.STM_Status.Status/TxPDO_Toggle <-> STM Status/Status/TxPDO Toggle
//     PlcTask Outputs/GVL_iXlinker.EtherCAT_Master_EJxxxx.Beckhoff_EJ7xxx.A_0003_EJ7041_0052_0016.ENC_Control_compact.Control/Enable_latch_extern_on_positive_edge <-> ENC Control compact/Control/Enable latch extern on positive edge
//     PlcTask Outputs/GVL_iXlinker.EtherCAT_Master_EJxxxx.Beckhoff_EJ7xxx.A_0003_EJ7041_0052_0016.ENC_Control_compact.Control/Set_counter <-> ENC Control compact/Control/Set counter
//     PlcTask Outputs/GVL_iXlinker.EtherCAT_Master_EJxxxx.Beckhoff_EJ7xxx.A_0003_EJ7041_0052_0016.ENC_Control_compact.Control/Enable_latch_extern_on_negative_edge <-> ENC Control compact/Control/Enable latch extern on negative edge
//     PlcTask Outputs/GVL_iXlinker.EtherCAT_Master_EJxxxx.Beckhoff_EJ7xxx.A_0003_EJ7041_0052_0016.ENC_Control_compact.Set_counter_value <-> ENC Control compact/Set counter value
//     PlcTask Outputs/GVL_iXlinker.EtherCAT_Master_EJxxxx.Beckhoff_EJ7xxx.A_0003_EJ7041_0052_0016.STM_Control.Control/Enable <-> STM Control/Control/Enable
//     PlcTask Outputs/GVL_iXlinker.EtherCAT_Master_EJxxxx.Beckhoff_EJ7xxx.A_0003_EJ7041_0052_0016.STM_Control.Control/Reset <-> STM Control/Control/Reset
//     PlcTask Outputs/GVL_iXlinker.EtherCAT_Master_EJxxxx.Beckhoff_EJ7xxx.A_0003_EJ7041_0052_0016.STM_Control.Control/Reduce_torque <-> STM Control/Control/Reduce torque
//     PlcTask Outputs/GVL_iXlinker.EtherCAT_Master_EJxxxx.Beckhoff_EJ7xxx.A_0003_EJ7041_0052_0016.STM_Velocity.Velocity <-> STM Velocity/Velocity
//     PlcTask Inputs/GVL_iXlinker.EtherCAT_Master_EJxxxx.Beckhoff_EJ7xxx.A_0003_EJ7041_0052_0016.WcState.WcState <-> WcState/WcState
//     PlcTask Inputs/GVL_iXlinker.EtherCAT_Master_EJxxxx.Beckhoff_EJ7xxx.A_0003_EJ7041_0052_0016.WcState.InputToggle <-> WcState/InputToggle
//     PlcTask Inputs/GVL_iXlinker.EtherCAT_Master_EJxxxx.Beckhoff_EJ7xxx.A_0003_EJ7041_0052_0016.InfoData.AdsAddr <-> InfoData/AdsAddr
//     PlcTask Inputs/GVL_iXlinker.EtherCAT_Master_EJxxxx.Beckhoff_EJ7xxx.A_0003_EJ7041_0052_0016.InfoData.Chn0 <-> InfoData/Chn0
//     PlcTask Inputs/GVL_iXlinker.EtherCAT_Master_EJxxxx.Beckhoff_EJ7xxx.A_0003_EJ7041_0052_0016.InfoData.Chn1 <-> InfoData/Chn1
//     PlcTask Inputs/GVL_iXlinker.EtherCAT_Master_EJxxxx.Beckhoff_EJ7xxx.A_0003_EJ7041_0052_0016.InfoData.State <-> InfoData/State
//   PLC/PLC Instance <-> EtherCAT Master EJxxxx/Beckhoff EJ7xxx/A_0004(EJ7047-0000-0018)
//     PlcTask Inputs/GVL_iXlinker.EtherCAT_Master_EJxxxx.Beckhoff_EJ7xxx.A_0004_EJ7047_0000_0018.ENC_Status_compact.Status/Latch_C_valid <-> ENC Status compact/Status/Latch C valid
//     PlcTask Inputs/GVL_iXlinker.EtherCAT_Master_EJxxxx.Beckhoff_EJ7xxx.A_0004_EJ7047_0000_0018.ENC_Status_compact.Status/Latch_extern_valid <-> ENC Status compact/Status/Latch extern valid
//     PlcTask Inputs/GVL_iXlinker.EtherCAT_Master_EJxxxx.Beckhoff_EJ7xxx.A_0004_EJ7047_0000_0018.ENC_Status_compact.Status/Set_counter_done <-> ENC Status compact/Status/Set counter done
//     PlcTask Inputs/GVL_iXlinker.EtherCAT_Master_EJxxxx.Beckhoff_EJ7xxx.A_0004_EJ7047_0000_0018.ENC_Status_compact.Status/Counter_underflow <-> ENC Status compact/Status/Counter underflow
//     PlcTask Inputs/GVL_iXlinker.EtherCAT_Master_EJxxxx.Beckhoff_EJ7xxx.A_0004_EJ7047_0000_0018.ENC_Status_compact.Status/Counter_overflow <-> ENC Status compact/Status/Counter overflow
//     PlcTask Inputs/GVL_iXlinker.EtherCAT_Master_EJxxxx.Beckhoff_EJ7xxx.A_0004_EJ7047_0000_0018.ENC_Status_compact.Status/Extrapolation_stall <-> ENC Status compact/Status/Extrapolation stall
//     PlcTask Inputs/GVL_iXlinker.EtherCAT_Master_EJxxxx.Beckhoff_EJ7xxx.A_0004_EJ7047_0000_0018.ENC_Status_compact.Status/Status_of_input_A <-> ENC Status compact/Status/Status of input A
